(* CODESYS project SPT_Diagnostic.library
   Author: SPT
   Version: 4.0.1
   Title: SPT Diagnostic
   DefaultNamespace: SPT_Diagnostic
   Placeholder: SPT Diagnostic
   Company: Beckhoff Automation LLC

Project tree, tasks and I/O mapping:
  libraries: SPT Base Types, * (Beckhoff Automation LLC); SPT Event Logger, * (Beckhoff Automation LLC); Tc2_EtherCAT, * (Beckhoff Automation GmbH); Tc2_IoFunctions, * (Beckhoff Automation GmbH); Tc2_Standard, * (Beckhoff Automation GmbH); Tc2_System, * (Beckhoff Automation GmbH); Tc2_Utilities, * (Beckhoff Automation GmbH); Tc3_EventLogger, * (Beckhoff Automation GmbH); Tc3_Module, * (Beckhoff Automation GmbH)
  Device Diagnostic/
    DUT/
      data type ST_DeviceInfo
    function block FB_Component_Devices [ST]: Reset, CyclicLogic, CyclicLogic_EtherCat, Update, Initialize, DeviceInfo, LocalAmsNetId
  EtherCat Diagnostic/
    DUT/
      data type ST_EtherCatMaster_Command
      data type ST_EtherCatMaster_Config
      data type ST_EtherCatMaster_HMI
      data type ST_EtherCatMaster_Status
      data type ST_SyncUnitInfo
    function F_EtherCAT_VendorIDtoString [ST]
    function block FB_EtherCatMaster [ST]: CreateEvents, Monitoring, Reset, CyclicLogic, Update, GetSlaveNameByAddr, GetSyncUnitSlaveNames, LookupMasterDevState, LookupSlaveDevState, RaiseAlarmWithStringsAndFlags, RaiseWarningWithStringParameters, SlaveIsPartOfSyncUnit, FB_init, HMICommunication, Initialize, MasterState, SlaveState, EtherCatMasterInfo
    function block FB_EtherCatSyncUnits [ST]: CyclicLogic, SyncUnits, Update, LocalAmsNetId
  Interface/
    interface I_Diagnostic: Update
    interface I_EtherCatSyncUnits: SyncUnits
    interface I_SafetyBase: DependenceFB, OK, SafetyReset
    interface I_SafetyReset: Execute, PulseDuration
    interface I_SafetySimulation: SimulateSafetyDiag, SimulateSafetyState
  Project Information/
    function F_GetCompany [ST]
    function F_GetTitle [ST]
    function F_GetVersion [ST]
  Safety/
    Safety FBs Diagnostic/
      DUT/
        data type E_ComponentSafetyConnection_State
        data type E_ComponentSafetyEdm_State
        data type E_ComponentSafetyEStop_State
        data type E_ComponentSafetyGroup_Diag
        data type E_ComponentSafetyGroup_State
        data type E_ComponentSafetyMon_State
        data type E_ComponentSafetyOrAnd_State
        data type ST_SafetyStateDiag
      Reset Functionblocks/
        function block FB_SafetyResetPulse [ST]: CyclicLogic, Execute, PulseDuration
      function block FB_Component_Safety_AndOrFB [ST]: CyclicLogic, Initialize
      function block FB_Component_Safety_Base [ST]: Reset, CyclicLogic, DependenceFB, OK, SafetyReset, SimulateSafetyDiag, SimulateSafetyState, Initialize
      function block FB_Component_Safety_ConnectionFB [ST]: CreateEvents, Monitoring, Reset, CyclicLogic, Initialize
      function block FB_Component_Safety_EdmFB [ST]: CreateEvents, Monitoring, Reset, CyclicLogic, Initialize
      function block FB_Component_Safety_EstopFB [ST]: CreateEvents, Monitoring, Reset, CyclicLogic, ActiveName, Initialize
      function block FB_Component_Safety_Group [ST]: CreateEvents, Monitoring, Reset, CyclicLogic, AutoResetConnectionFaults, Initialize
      function block FB_Component_Safety_MonFB [ST]: CreateEvents, Monitoring, Reset, CyclicLogic, ActiveAlarm, ActiveName
    Safety Hardware Diagnostic/
  Version/
    global variables Global_Version
  00000000-0000-0000-0000-000000000000|LICENSE
  LICENSE
  global variables Parameter_Diagnostic
*)

// Device Diagnostic/DUT/ST_DeviceInfo
TYPE ST_DeviceInfo :
	STRUCT
		AmsNetID	   : T_AMSNETID;
		DeviceID	   : UINT;
		DeviceName	   : T_MAXSTRING;
		DeviceType	   : IODEVICETYPES;
		ipDiagnosticFB : I_Diagnostic;
	END_STRUCT
END_TYPE

// EtherCat Diagnostic/DUT/ST_EtherCatMaster_Command
TYPE ST_EtherCatMaster_Command :
	STRUCT
	END_STRUCT
END_TYPE

// EtherCat Diagnostic/DUT/ST_EtherCatMaster_Config
TYPE ST_EtherCatMaster_Config :
	STRUCT
		DeviceInfo : ST_DeviceInfo;
	END_STRUCT
END_TYPE

// EtherCat Diagnostic/DUT/ST_EtherCatMaster_HMI
TYPE ST_EtherCatMaster_HMI :
	STRUCT
		Config	: ST_EtherCatMaster_Config;
		Command : ST_EtherCatMaster_Command;
		Status	: ST_EtherCatMaster_Status;
	END_STRUCT
END_TYPE

// EtherCat Diagnostic/DUT/ST_EtherCatMaster_Status
TYPE ST_EtherCatMaster_Status :
	STRUCT
		EcSlavesState		: ARRAY[0..Parameter_Diagnostic.ETHERCAT_MASTER_SLAVE_MAX] OF ST_EcSlaveState;
		ConfiguredSlaveInfo : ARRAY[0..Parameter_Diagnostic.ETHERCAT_MASTER_SLAVE_MAX] OF ST_EcSlaveConfigData;
		EcSlaveTopologyInfo : ARRAY[0..Parameter_Diagnostic.ETHERCAT_MASTER_SLAVE_MAX] OF ST_TopologyDataEx;
	END_STRUCT
END_TYPE

// EtherCat Diagnostic/DUT/ST_SyncUnitInfo
TYPE ST_SyncUnitInfo :
	STRUCT
		Parent		   : T_MAXSTRING;
		Name		   : STRING(63);
		NumberOfSlaves : UINT;
		Slaves		   : ARRAY[1..Parameter_Diagnostic.ETHERCAT_MASTER_SYNC_UNIT_SLAVE_MAX] OF UINT;
	END_STRUCT
END_TYPE

// Safety/Safety FBs Diagnostic/DUT/E_ComponentSafetyConnection_State
{attribute 'qualified_only'}
{attribute 'strict'}
TYPE E_ComponentSafetyConnection_State : (
		Reset	   := 100,
		Session	   := 101,
		Connection := 102,
		Parameter  := 103,
		Data	   := 104,
		Shutdown   := 105,
		Deactive   := 106
	) USINT;
END_TYPE

// Safety/Safety FBs Diagnostic/DUT/E_ComponentSafetyEdm_State
{attribute 'qualified_only'}
TYPE E_ComponentSafetyEdm_State : (
		Invalid := 0,
		Stop	:= 2,
		Error	:= 4,
		Reset	:= 5,
		MonOff	:= 14,
		MonOn	:= 15
	) USINT;
END_TYPE

// Safety/Safety FBs Diagnostic/DUT/E_ComponentSafetyEStop_State
{attribute 'qualified_only'}
TYPE E_ComponentSafetyEStop_State : (
		Invalid	 := 0,
		Run		 := 1,
		Stop	 := 2,
		Safe	 := 3,
		Error	 := 4,
		Reset	 := 5,
		Start	 := 6,
		DelayOut := 7
	) USINT;
END_TYPE

// Safety/Safety FBs Diagnostic/DUT/E_ComponentSafetyGroup_Diag
{attribute 'qualified_only'}
TYPE E_ComponentSafetyGroup_Diag : (
		NoError		  := 0,
		FbError		  := 1,
		ComError	  := 2,
		ModuleError	  := 3,
		CmpError	  := 4,
		DeactiveError := 5,
		RestartError  := 6
	) UINT;
END_TYPE

// Safety/Safety FBs Diagnostic/DUT/E_ComponentSafetyGroup_State
{attribute 'qualified_only'}
TYPE E_ComponentSafetyGroup_State : (
		Invalid		 := 0,
		Run			 := 1,
		Stop		 := 2,
		Error		 := 4,
		Reset		 := 5,
		Start		 := 6,
		StopError	 := 7,
		Deactive	 := 16,
		WaitComError := 17
	) USINT;
END_TYPE

// Safety/Safety FBs Diagnostic/DUT/E_ComponentSafetyMon_State
{attribute 'qualified_only'}
TYPE E_ComponentSafetyMon_State : (
		Invalid	   := 0,
		Run		   := 1,
		Stop	   := 2,
		Safe	   := 3,
		Error	   := 4,
		Reset	   := 5,
		Start	   := 6,
		ErrorDelay := 7,
		DelayOut   := 8,
		FuncTest   := 9
	) USINT;
END_TYPE

// Safety/Safety FBs Diagnostic/DUT/E_ComponentSafetyOrAnd_State
{attribute 'qualified_only'}
TYPE E_ComponentSafetyOrAnd_State : (
		Invalid := 0,
		Run		:= 1,
		Stop	:= 2,
		Safe	:= 3
	) USINT;
END_TYPE

// Safety/Safety FBs Diagnostic/DUT/ST_SafetyStateDiag
{attribute 'pack_mode' := '1'}
TYPE ST_SafetyStateDiag :
	STRUCT
		State : USINT;
		Diag  : UINT; // **NOT PRESENT ON AND/OR FBs ** For components with USINT as Diag connection, connect first 8 Bit of UINT Diag. Inherited FB is evaluating correct length.
	END_STRUCT
END_TYPE

// Version/Global_Version
{attribute 'TcGenerated'}
{attribute 'no-analysis'}
{attribute 'linkalways'}
// This function has been automatically generated from the project information.
VAR_GLOBAL CONSTANT
	{attribute 'const_non_replaced'}
	stLibVersion_SPT_Diagnostic : ST_LibVersion := (iMajor := 4, iMinor := 0, iBuild := 1, iRevision := 0, nFlags := 0, sVersion := '4.0.1');
END_VAR

// Parameter_Diagnostic
{attribute 'qualified_only'}
VAR_GLOBAL CONSTANT
	UPDATE_TIME : TIME	:= T#500MS; // Start Diagnostic Run every xxx ms, T#0s = deactivated, update needs to manually occur via I_Diagnostic.Upadate()
	DEVICES_MAX : UDINT := 5;		// Max Devices in this System

	// EtherCat
	ETHERCAT_MASTER_START_UP_TIME		: TIME					  := T#1S; // Time to Startup EtherCat Master Diagnostic at initial startup
	ETHERCAT_MASTER_MAX					: UDINT					  := 5;	   // Max EtherCat Masters
	ETHERCAT_MASTER_SLAVE_MAX			: UDINT(1..EC_MAX_SLAVES) := 50;   // Max Slaves per EtherCat Master
	ETHERCAT_MASTER_SYNC_UNIT_MAX		: UDINT					  := 10;   // Max Count of Sync Units per Master
	ETHERCAT_MASTER_SYNC_UNIT_SLAVE_MAX : UDINT					  := 30;   // Max Count of Slaves per Sync Unit
END_VAR

// Device Diagnostic/FB_Component_Devices
{attribute 'no_explicit_call' := 'do not call this FB directly'}
FUNCTION_BLOCK FB_Component_Devices EXTENDS FB_ComponentBase IMPLEMENTS I_Diagnostic
VAR
	// System Information
	GetLocalAmsNetId : FB_GetLocalAmsNetId;
	GetDeviceIds	 : IOF_GetDeviceIDs;
	DeviceIds		 : ARRAY[0..Parameter_Diagnostic.DEVICES_MAX] OF WORD; // 0 = Device counter, 1..X = Device ID's
	GetDeviceType	 : IOF_GetDeviceType;
	GetDeviceName	 : IOF_GetDeviceName;
	GetDeviceNetId	 : IOF_GetDeviceNetId;

	// Instances of Devices
	EtherCatSyncUnits	: FB_EtherCatSyncUnits;																		  // All Sync Units in this runtime
	EtherCatMaster		: ARRAY[1..Parameter_Diagnostic.ETHERCAT_MASTER_MAX] OF FB_EtherCatMaster(EtherCatSyncUnits); //
	EtherCatMasterCount : UDINT(0..Parameter_Diagnostic.ETHERCAT_MASTER_MAX) := 0;									  // Start at 0 to identify existing during Initialzation

	// Properties
	_DeviceInfo	   : ARRAY[1..Parameter_Diagnostic.DEVICES_MAX] OF ST_DeviceInfo;
	_LocalAmsNetId : T_AmsNetId := '';

	// Alarms

	// HMI

	// Sequences
	InitializeSequence : UDINT := 0;
	DeviceNumber	   : UDINT := 1;
	i				   : UDINT := 0; // Iterator
END_VAR

VAR
	// Local
	UpdateOn	: TON;
	UpdateOff	: TON;
	RtrigUpdate : R_TRIG;
END_VAR

// Clears error flags and error IDs for this component
METHOD PUBLIC Reset : BOOL
Reset := SUPER^.Reset();
IF EtherCatMasterCount >= 1 THEN
	FOR i := 1 TO EtherCatMasterCount DO
		EtherCatMaster[i].Reset();
	END_FOR
END_IF
END_METHOD

// This method serves as the entry point for all underlying FB logic
METHOD PUBLIC CyclicLogic

// This method should be called cyclically by descendant function blocks by invoking SUPER^.CyclicLogic().  Alternatively, the contents of this method could be reimplemented entirely in which case a call to this method would not be necessary.
IF NOT _InitComplete THEN
	_InitComplete := Initialize();
	RETURN;
END_IF

// Update Toggle
IF Parameter_Diagnostic.UPDATE_TIME > T#0MS THEN
	UpdateOn(IN := NOT UpdateOff.Q, PT := Parameter_Diagnostic.UPDATE_TIME);
	UpdateOff(IN := UpdateOn.Q, PT := Parameter_Diagnostic.UPDATE_TIME);
	RtrigUpdate(CLK := UpdateOn.Q);
END_IF

// Cyclic Logics
CyclicLogic_EtherCat();
SUPER^.CyclicLogic();

// Error Status Update of all Devices
_Error := FALSE;
_Busy  := FALSE;
IF EtherCatMasterCount >= 1 THEN
	FOR i := 1 TO EtherCatMasterCount DO
		IF _CurrentAlarmSeverity < EtherCatMaster[i].CurrentAlarmSeverity THEN
			_CurrentAlarmSeverity := EtherCatMaster[i].CurrentAlarmSeverity;
		END_IF

		_Error := _Error OR EtherCatMaster[i].Error;
		_Busy  := _Busy OR EtherCatMaster[i].Busy;
		IF EtherCatMaster[i].ErrorID <> 0 AND _ErrorID = 0 THEN
			_ErrorID := EtherCatMaster[i].ErrorID;
		END_IF
	END_FOR
END_IF
END_METHOD

METHOD CyclicLogic_EtherCat
// Get all Sync Units in Runtime
EtherCatSyncUnits.LocalAmsNetId := _LocalAmsNetId;
EtherCatSyncUnits.CyclicLogic();

// Call Cyclic
IF EtherCatMasterCount >= 1 THEN
	FOR i := 1 TO EtherCatMasterCount DO
		// Update
		IF RtrigUpdate.Q THEN
			EtherCatMaster[i].Update();
		END_IF

		// Cyclic Call
		EtherCatMaster[i].CyclicLogic();
	END_FOR
END_IF
END_METHOD

METHOD Update
IF EtherCatMasterCount >= 1 THEN
	FOR i := 1 TO EtherCatMasterCount DO
		EtherCatMaster[i].Update();
	END_FOR
END_IF
END_METHOD

// Basic component initialization logic
METHOD PROTECTED Initialize : BOOL;
// This method is called by CyclicLogic() as required
VAR_INST
	AllDevicesInitialized : BOOL := FALSE;
END_VAR
Initialize := FALSE;
IF _Simulate THEN
	Initialize := SUPER^.Initialize();
	RETURN;
END_IF

// Call FBs
GetLocalAmsNetId(tTimeOut := T#1S);
GetDeviceIds(NETID := _LocalAmsNetId, TMOUT := T#1S);
GetDeviceName(NETID := _LocalAmsNetId, TMOUT := T#1S);
GetDeviceNetId(NETID := _LocalAmsNetId, TMOUT := T#1S);
GetDeviceType(NETID := _LocalAmsNetId, TMOUT := T#1S);

// Init Sequence
CASE InitializeSequence OF
	0: // Get local AmsNet-Id
		GetLocalAmsNetId.bExecute := TRUE;
		IF GetLocalAmsNetId.bBusy THEN
			InitializeSequence := InitializeSequence + 10;
		END_IF

	10: // Get local AmsNet-Id
		IF NOT GetLocalAmsNetId.bBusy AND NOT GetLocalAmsNetId.bError THEN
			_LocalAmsNetId	   := GetLocalAmsNetId.AddrString;
			InitializeSequence := InitializeSequence + 10;
		END_IF

		IF GetLocalAmsNetId.bError THEN
			_ErrorID := GetLocalAmsNetId.nErrId;
			Trace('Init Failed - GetLocalAmsNetId!');
			InitializeSequence := 999;
		END_IF

	20: // Get all Devices in this System
		GetDeviceIds.LEN	  := SIZEOF(DeviceIds);
		GetDeviceIds.DESTADDR := ADR(DeviceIds);
		GetDeviceIds.START	  := TRUE;
		IF GetDeviceIds.BUSY THEN
			GetDeviceIds.START := FALSE;
			InitializeSequence := InitializeSequence + 10;
		END_IF

	30: // Get all Devices in this System
		IF NOT GetDeviceIds.BUSY AND NOT GetDeviceIds.ERR THEN
			// Devices found
			IF (DeviceIDs[0] > 0) AND NOT _Simulate THEN
				// Map device Ids
				FOR i := 1 TO DeviceIDs[0] DO
					IF i <= Parameter_Diagnostic.DEVICES_MAX THEN
						_DeviceInfo[i].DeviceID := DeviceIDs[i];
					ELSE
						Trace('Init Failed - find IO Devices, Diagnostic, not enough Devices foreseen! Increase DEVICES_MAX');
						InitializeSequence := 999;
						EXIT;
					END_IF
				END_FOR

				InitializeSequence := InitializeSequence + 10;
			ELSE
				_Simulate		   := TRUE; // No devices found = activate simulation mode
				InitializeSequence := 1000;
			END_IF
		END_IF

		IF GetDeviceIds.ERR THEN
			_ErrorID := GetDeviceIds.ERRID;
			Trace('Init Failed - GetDeviceIds!');
			InitializeSequence := 999;
		END_IF

	40: // Get Device Names
		GetDeviceName.DEVICEID := DeviceIDs[DeviceNumber];
		GetDeviceName.START	   := TRUE;
		IF GetDeviceName.BUSY THEN
			GetDeviceName.START := FALSE;
			InitializeSequence	:= InitializeSequence + 10;
		END_IF

	50: // Get Device Names
		IF NOT GetDeviceName.BUSY AND NOT GetDeviceName.ERR THEN
			// Next Device
			_DeviceInfo[DeviceNumber].DeviceName := GetDeviceName.DEVICENAME;
			DeviceNumber						 := DeviceNumber + 1;
			IF (DeviceIDs[DeviceNumber] <> 0) THEN
				InitializeSequence := InitializeSequence - 10;
			ELSE
				DeviceNumber	   := 1;
				InitializeSequence := InitializeSequence + 10;
			END_IF
		END_IF

		IF GetDeviceName.ERR THEN
			_ErrorID := GetDeviceName.ERRID;
			Trace('Init Failed - GetDeviceName!');
			InitializeSequence := 999;
		END_IF

	60: // Get Device NetIds
		GetDeviceNetId.DEVICEID := DeviceIDs[DeviceNumber];
		GetDeviceNetId.START	:= TRUE;
		IF GetDeviceNetId.BUSY THEN
			GetDeviceNetId.START := FALSE;
			InitializeSequence	 := InitializeSequence + 10;
		END_IF

	70: // Get Device NetIds
		IF NOT GetDeviceNetId.BUSY AND NOT GetDeviceNetId.ERR THEN
			// Next Device
			_DeviceInfo[DeviceNumber].AmsNetID := GetDeviceNetId.DeviceNetId;
			DeviceNumber					   := DeviceNumber + 1;
			IF (DeviceIDs[DeviceNumber] <> 0) THEN
				InitializeSequence := InitializeSequence - 10;
			ELSE
				DeviceNumber	   := 1;
				InitializeSequence := InitializeSequence + 10;
			END_IF
		END_IF

		IF GetDeviceNetId.ERR THEN
			_ErrorID := GetDeviceNetId.ERRID;
			Trace('Init Failed - GetDeviceNetId!');
			InitializeSequence := 999;
		END_IF

	80: // Get Device Types
		GetDeviceType.DEVICEID := DeviceIDs[DeviceNumber];
		GetDeviceType.START	   := TRUE;
		IF GetDeviceType.BUSY THEN
			GetDeviceType.START := FALSE;
			InitializeSequence	:= InitializeSequence + 10;
		END_IF

	90: // Get Device Types
		IF NOT GetDeviceType.BUSY AND NOT GetDeviceType.ERR THEN
			// Next Device
			_DeviceInfo[DeviceNumber].DeviceType := GetDeviceType.IODeviceType;
			DeviceNumber						 := DeviceNumber + 1;
			IF (DeviceIDs[DeviceNumber] <> 0) THEN
				InitializeSequence := InitializeSequence - 10;
			ELSE
				DeviceNumber	   := 1;
				InitializeSequence := InitializeSequence + 10;
			END_IF
		END_IF

		IF GetDeviceType.ERR THEN
			_ErrorID := GetDeviceType.ERRID;
			Trace('Init Failed - GetDeviceType!');
			InitializeSequence := 999;
		END_IF

	100: // Initalize all Devices found
		FOR i := 1 TO DeviceIDs[0] DO
			CASE DeviceInfo[i].DeviceType OF
				IODEVICETYPES.IODEVICETYPE_ETHERCAT:
					EtherCatMasterCount := EtherCatMasterCount + 1;
					IF EtherCatMasterCount <= Parameter_Diagnostic.ETHERCAT_MASTER_MAX THEN
						EtherCatMaster[EtherCatMasterCount].EtherCatMasterInfo REF= _DeviceInfo[i];
						EtherCatMaster[EtherCatMasterCount].Name			   := DeviceInfo[i].DeviceName;
						DeviceInfo[i].ipDiagnosticFB						   := EtherCatMaster[EtherCatMasterCount];
					ELSE
						Trace('Init Failed - not enough EtherCat Master Diagnostics Instances! Increase ETHERCAT_MASTER_MAX');
						InitializeSequence := 999;
					END_IF

			ELSE
				Trace(CONCAT('Warning - Device Diagnostics for this Device does not exist! ', DeviceInfo[i].DeviceName));
			END_CASE
		END_FOR

		// No error during initialization
		IF InitializeSequence <> 999 THEN
			InitializeSequence := InitializeSequence + 10;
		END_IF

	110: // Initalize all Devices found
		AllDevicesInitialized := TRUE;

		// Init all EtherCat Master Devices
		IF EtherCatMasterCount >= 1 THEN
			FOR i := 1 TO EtherCatMasterCount DO
				EtherCatMaster[i].CyclicLogic();
				AllDevicesInitialized := AllDevicesInitialized AND EtherCatMaster[i].InitComplete;
			END_FOR
		END_IF

		IF AllDevicesInitialized THEN
			InitializeSequence := 1000;
		END_IF

	1000: // Initialize the Base
		IF SUPER^.Initialize() THEN
			Initialize := TRUE;
			_Error	   := FALSE;
			_Busy	   := FALSE;
		END_IF

	999:
		_Error := TRUE;
		_Busy  := FALSE;
END_CASE
END_METHOD

{analysis -29}
PROPERTY DeviceInfo : REFERENCE TO ARRAY[1..Parameter_Diagnostic.DEVICES_MAX] OF ST_DeviceInfo
GET
DeviceInfo REF= _DeviceInfo;
END_GET
END_PROPERTY

PROPERTY LocalAmsNetId : T_AmsNetId
GET
LocalAmsNetId := _LocalAmsNetId;
END_GET
END_PROPERTY

END_FUNCTION_BLOCK

// Interface/I_Diagnostic
INTERFACE I_Diagnostic EXTENDS I_BaseFB

METHOD Update
VAR_INPUT
END_VAR
END_METHOD

END_INTERFACE

// EtherCat Diagnostic/FB_EtherCatSyncUnits
{attribute 'no_explicit_call' := 'do not call this FB directly'}
FUNCTION_BLOCK FB_EtherCatSyncUnits EXTENDS FB_CyclicFB IMPLEMENTS I_EtherCatSyncUnits
VAR
	(* Sequence *)
	SyncUnitSequence : UINT;

	(* Local *)
	GetSyncUnitOids			  : ADSRDWRT;
	GetAllSyncUnitSlaveAddr	  : FB_EcGetAllSyncUnitSlaveAddr;
	ipSyncUnitComObject		  : ITComObject;
	ipSyncUnitParentComObject : ITComObject;
	SyncUnitCount			  : DWORD;
	i						  : DWORD; // Iterator
	SyncUnitParentOid		  : OTCID;
	SyncUnitOids			  : ARRAY[1..Parameter_Diagnostic.ETHERCAT_MASTER_SYNC_UNIT_MAX] OF OTCID;

	(* Properties *)
	_SyncUnits	   : ARRAY[1..Parameter_Diagnostic.ETHERCAT_MASTER_SYNC_UNIT_MAX] OF ST_SyncUnitInfo;
	_LocalAmsNetId : T_AmsNetId;
END_VAR

VAR CONSTANT
	SYNC_UNIT_CLASS_ID : CLSID := STRING_TO_GUID('03020004-0000-0000-F000-000000000064');
END_VAR

METHOD PUBLIC CyclicLogic
VAR_INST
	tempName		 : STRING(63);
	SyncUnitIterator : UINT := 1;
END_VAR
{analysis -19}
{analysis -07}

// Call FBs
GetSyncUnitOids(NETID := _LocalAmsNetId);
GetAllSyncUnitSlaveAddr(sNetId := _LocalAmsNetId);

// Sequence
CASE SyncUnitSequence OF
	0: // Wait for start
		GetSyncUnitOids.WRTRD			 := FALSE;
		GetAllSyncUnitSlaveAddr.bExecute := FALSE;
		SyncUnitIterator				 := 1;

	10: // Get Sync Unit Count

		// Reset for restart
		_Error	 := FALSE;
		_ErrorID := 0;

		// Get Sync Unit Count
		GetSyncUnitOids.PORT	 := 10;
		GetSyncUnitOids.IDXGRP	 := 16#201;
		GetSyncUnitOids.IDXOFFS	 := 16#01;
		GetSyncUnitOids.WRITELEN := SIZEOF(SYNC_UNIT_CLASS_ID);
		GetSyncUnitOids.SRCADDR	 := ADR(SYNC_UNIT_CLASS_ID);
		GetSyncUnitOids.READLEN	 := SIZEOF(SyncUnitCount);
		GetSyncUnitOids.DESTADDR := ADR(SyncUnitCount);
		GetSyncUnitOids.WRTRD	 := TRUE;
		IF GetSyncUnitOids.BUSY THEN
			SyncUnitSequence := SyncUnitSequence + 10;
		END_IF

	20: // Get Sync Unit Count
		IF NOT GetSyncUnitOids.BUSY AND NOT GetSyncUnitOids.ERR THEN
			// Byte Adjustment
			SyncUnitCount		  := SyncUnitCount / 4;
			GetSyncUnitOids.WRTRD := FALSE;
			IF SyncUnitCount <= Parameter_Diagnostic.ETHERCAT_MASTER_SYNC_UNIT_MAX THEN // Check configuration and space
				IF SyncUnitCount > 0 THEN												// Only if Sync Unit exist - run diag
					SyncUnitSequence := SyncUnitSequence + 10;
				ELSE
					SyncUnitSequence := 0;
				END_IF
			ELSE
				SyncUnitSequence := 999;
				_ErrorID		 := SyncUnitCount;
				Trace('FB_EtherCatSyncUnits - not enough Sync Units foreseen! Increase ETHERCAT_MASTER_SYNC_UNIT_MAX');
			END_IF
		END_IF

		IF GetSyncUnitOids.ERR THEN
			_ErrorID		 := GetSyncUnitOids.ERRID;
			SyncUnitSequence := 999;
		END_IF

	30: // Get Sync Unit Oids
		GetSyncUnitOids.PORT	 := 10;
		GetSyncUnitOids.IDXGRP	 := 16#201;
		GetSyncUnitOids.IDXOFFS	 := 16#02;
		GetSyncUnitOids.WRITELEN := SIZEOF(SYNC_UNIT_CLASS_ID);
		GetSyncUnitOids.SRCADDR	 := ADR(SYNC_UNIT_CLASS_ID);
		GetSyncUnitOids.READLEN	 := (SIZEOF(OTCID) * SyncUnitCount);
		GetSyncUnitOids.DESTADDR := ADR(SyncUnitOids);
		GetSyncUnitOids.WRTRD	 := TRUE;
		IF GetSyncUnitOids.BUSY THEN
			SyncUnitSequence := SyncUnitSequence + 10;
		END_IF

	40: // Get Sync Unit Oids
		IF NOT GetSyncUnitOids.BUSY AND NOT GetSyncUnitOids.ERR THEN
			GetSyncUnitOids.WRTRD := FALSE;
			SyncUnitSequence	  := SyncUnitSequence + 10;
		END_IF

		IF GetSyncUnitOids.ERR THEN
			_ErrorID		 := GetSyncUnitOids.ERRID;
			SyncUnitSequence := 999;
		END_IF

	50: // Get EtherCat Master and Name of Sync Unit
		FOR i := 1 TO SyncUnitCount DO
			// Get Sync Unit
			FW_ObjMgr_GetObjectInstance(SyncUnitOids[i], TC_GLOBAL_IID_LIST.IID_ITComObject, ADR(ipSyncUnitComObject));
			IF ipSyncUnitComObject <> 0 THEN
				ipSyncUnitComObject.TcGetObjectName(objName := ADR(_SyncUnits[i].Name), nameLen := SIZEOF(_SyncUnits[i].Name));
				F_EcGetSyncUnitName(SyncUnitOids[i], sSyncUnitName => tempName);
				tempName		   := CONCAT(tempName, ' - ');
				_SyncUnits[i].Name := CONCAT(tempName, _SyncUnits[i].Name);

				// Get Parent
				ipSyncUnitComObject.TcGetParentObjId(SyncUnitParentOid);
				FW_ObjMgr_GetObjectInstance(SyncUnitParentOid, TC_GLOBAL_IID_LIST.IID_ITComObject, ADR(ipSyncUnitParentComObject));
				IF ipSyncUnitParentComObject <> 0 THEN
					ipSyncUnitParentComObject.TcGetObjectName(objName := ADR(_SyncUnits[i].Parent), nameLen := SIZEOF(_SyncUnits[i].Parent));
					FW_SafeRelease(pipUnk := ADR(ipSyncUnitParentComObject));
				END_IF

				FW_SafeRelease(pipUnk := ADR(ipSyncUnitComObject));
			END_IF
		END_FOR

		SyncUnitSequence := SyncUnitSequence + 10;

	60: // Get all sync Unit Slaves 
		IF SyncUnitIterator > Parameter_Diagnostic.ETHERCAT_MASTER_SYNC_UNIT_MAX THEN
			SyncUnitSequence := 0; // All Sync units searched
		ELSE
			IF SyncUnitOids[SyncUnitIterator] = 0 THEN
				SyncUnitSequence := 0; // Done
			ELSE
				GetAllSyncUnitSlaveAddr.nObjectId := SyncUnitOids[SyncUnitIterator];
				GetAllSyncUnitSlaveAddr.pAddrBuf  := ADR(_SyncUnits[SyncUnitIterator].Slaves);
				GetAllSyncUnitSlaveAddr.cbBufLen  := SIZEOF(_SyncUnits[SyncUnitIterator].Slaves);
				GetAllSyncUnitSlaveAddr.bExecute  := TRUE;
				IF GetAllSyncUnitSlaveAddr.bBusy THEN
					GetAllSyncUnitSlaveAddr.bExecute := FALSE;
					SyncUnitSequence				 := SyncUnitSequence + 10;
				END_IF
			END_IF
		END_IF

	70: // Get all sync Unit Slaves
		IF NOT GetAllSyncUnitSlaveAddr.bBusy AND NOT GetAllSyncUnitSlaveAddr.bError THEN
			_SyncUnits[SyncUnitIterator].NumberOfSlaves := GetAllSyncUnitSlaveAddr.nSlaves;
			SyncUnitIterator							:= SyncUnitIterator + 1;
			IF _SyncUnits[SyncUnitIterator].NumberOfSlaves <= Parameter_Diagnostic.ETHERCAT_MASTER_SYNC_UNIT_SLAVE_MAX THEN
				SyncUnitSequence := SyncUnitSequence - 10;
			ELSE
				SyncUnitSequence := 999;
				_ErrorID		 := _SyncUnits[SyncUnitIterator].NumberOfSlaves;
				Trace('FB_EtherCatSyncUnits - not enough slaves per Sync Units foreseen! Increase ETHERCAT_MASTER_SYNC_UNIT_SLAVE_MAX');
			END_IF
		END_IF

		IF GetAllSyncUnitSlaveAddr.bError THEN
			_ErrorID		 := GetAllSyncUnitSlaveAddr.nErrId;
			SyncUnitSequence := 999;
		END_IF

	999: // Error
		SyncUnitSequence := 0;
		_Error			 := TRUE;
		Trace('FB_EtherCatSyncUnits - Error get Sync Units Sequence!');
END_CASE

_Busy := SyncUnitSequence <> 0;
END_METHOD

PROPERTY SyncUnits : REFERENCE TO ARRAY[1..Parameter_Diagnostic.ETHERCAT_MASTER_SYNC_UNIT_MAX] OF ST_SyncUnitInfo
GET
SyncUnits REF= _SyncUnits;
END_GET
END_PROPERTY

METHOD Update
IF NOT _Busy THEN
	SyncUnitSequence := 10;
END_IF
END_METHOD

PROPERTY LocalAmsNetId : T_AmsNetId
SET
_LocalAmsNetId := LocalAmsNetId;
END_SET
END_PROPERTY

END_FUNCTION_BLOCK

// Interface/I_EtherCatSyncUnits
INTERFACE I_EtherCatSyncUnits EXTENDS I_Diagnostic

PROPERTY SyncUnits : REFERENCE TO ARRAY[1..Parameter_Diagnostic.ETHERCAT_MASTER_SYNC_UNIT_MAX] OF ST_SyncUnitInfo
GET
END_GET
END_PROPERTY

END_INTERFACE

// EtherCat Diagnostic/FB_EtherCatMaster
{attribute 'no_explicit_call' := 'do not call this FB directly'}
FUNCTION_BLOCK FB_EtherCatMaster EXTENDS FB_ComponentBase IMPLEMENTS I_Diagnostic
VAR
	(* Internal Variables *)
	EcGetMasterDevState	 : FB_EcGetMasterDevState;
	GetSlaveTopologyInfo : FB_EcGetSlaveTopologyInfo;
	EcGetAllSlaveStates	 : FB_EcGetAllSlaveStates;
	GetConfiguredSlaves	 : FB_EcGetConfSlaves;
	EcSlavesState		 : ARRAY[0..Parameter_Diagnostic.ETHERCAT_MASTER_SLAVE_MAX] OF ST_EcSlaveState;
	ConfiguredSlaveInfo	 : ARRAY[0..Parameter_Diagnostic.ETHERCAT_MASTER_SLAVE_MAX] OF ST_EcSlaveConfigData;
	EcSlaveTopologyInfo	 : ARRAY[0..Parameter_Diagnostic.ETHERCAT_MASTER_SLAVE_MAX] OF ST_TopologyDataEx;
	SyncUnits			 : REFERENCE TO ARRAY[1..Parameter_Diagnostic.ETHERCAT_MASTER_SYNC_UNIT_MAX] OF ST_SyncUnitInfo;
	MasterDevState		 : WORD;
	SlaveCount			 : UINT;
	CfgSlaveCount		 : UINT;

	(* Properties *)
	_EtherCatMasterInfo : REFERENCE TO ST_DeviceInfo;

	(* HMI *)
	EtherCatMaster_HMI : ST_EtherCatMaster_HMI;

	(* Sync Units *)
	ipEtherCatSyncUnits : I_EtherCatSyncUnits;

	(* Sequence *)
	SlaveSeq	: UINT;
	MasterSeq	: UINT;
	SyncUnitSeq : UINT;

	(* Alarms *)
	MasterAlarms	 : ARRAY[1..MASTER_ALARM_COUNT] OF FB_TcAlarm;
	SlaveErrors		 : ARRAY[0..Parameter_Diagnostic.ETHERCAT_MASTER_SLAVE_MAX] OF FB_TcAlarm;
	SlaveWarnings	 : ARRAY[0..Parameter_Diagnostic.ETHERCAT_MASTER_SLAVE_MAX] OF FB_TcAlarm;
	SyncUnitWarnings : ARRAY[1..Parameter_Diagnostic.ETHERCAT_MASTER_SYNC_UNIT_MAX] OF FB_TcAlarm;
END_VAR

VAR CONSTANT
	MASTER_ALARM_COUNT : UDINT := 3;
	STRING_LEN		   : INT   := 80;
END_VAR

METHOD PROTECTED CreateEvents
// This method is called by Initialize() as required
VAR_INST
	tempName   : STRING;
	SourceInfo : FB_TcSourceInfo;
	i		   : UDINT;
END_VAR
F_CreateAllEventsInClass(Alarms		:= MasterAlarms,
						 ClassSize	:= SIZEOF(TC_EVENTS.EtherCatMaster),
						 pInitEvent := ADR(TC_EVENTS.EtherCatMaster.InitReferenceEvent),
						 Prefix		:= Name);

SUPER^.CreateEvents();

// Create SyncUnit and Slave Alarms
FOR i := 0 TO Parameter_Diagnostic.ETHERCAT_MASTER_SLAVE_MAX DO
	SourceInfo.sName := CONCAT(CONCAT(THIS^.Name, ' - '), ConfiguredSlaveInfo[i].sName);
	SlaveErrors[i].CreateEx(stEventEntry := TC_EVENTS.EtherCatSlave.SlaveError, 0, SourceInfo);
	SlaveWarnings[i].CreateEx(stEventEntry := TC_EVENTS.EtherCatSlave.SlaveWarning, 0, SourceInfo);
END_FOR

FOR i := 1 TO Parameter_Diagnostic.ETHERCAT_MASTER_SYNC_UNIT_MAX DO
	SourceInfo.sName := CONCAT(CONCAT(THIS^.Name, ' - '), ConfiguredSlaveInfo[i].sName);
	SyncUnitWarnings[i].CreateEx(stEventEntry := TC_EVENTS.SyncUnit.SyncUnitWarning, 0, SourceInfo);
END_FOR
END_METHOD

// Provides basic error detection and event handling for this component
METHOD PROTECTED Monitoring
// This method is called cyclically by CyclicLogic()
VAR_INST
	Error1 : BOOL;
	Error2 : BOOL;
	Error3 : BOOL;
END_VAR
SUPER^.Monitoring();

(* EtherCat Master Messages *)

// Raised in Master Sequence

(* EtherCat Slave Messages *)

// Raised in Slave Sequence

(* Alarm Severity of EtherCat Master Device *)
_CurrentAlarmSeverity := F_GetMaxSeverityRaised(Alarms := MasterAlarms, CurrentSeverity := _CurrentAlarmSeverity);
_CurrentAlarmSeverity := F_GetMaxSeverityRaised(Alarms := SlaveErrors, CurrentSeverity := _CurrentAlarmSeverity);
_CurrentAlarmSeverity := F_GetMaxSeverityRaised(Alarms := SlaveWarnings, CurrentSeverity := _CurrentAlarmSeverity);
_CurrentAlarmSeverity := F_GetMaxSeverityRaised(Alarms := SyncUnitWarnings, CurrentSeverity := _CurrentAlarmSeverity);
END_METHOD

// Clears error flags and error IDs for this component
METHOD PUBLIC Reset : BOOL
F_ClearAllEventsInClass(MasterAlarms);
F_ClearAllEventsInClass(SlaveErrors);
F_ClearAllEventsInClass(SlaveWarnings);
F_ClearAllEventsInClass(SyncUnitWarnings);
SlaveSeq  := 0;
MasterSeq := 0;
_Error	  := FALSE;
_ErrorID  := 0;
_Busy	  := FALSE;
Reset	  := SUPER^.Reset();
END_METHOD

// This method serves as the entry point for all underlying FB logic
METHOD PUBLIC CyclicLogic

// This method should be called cyclically by descendant function blocks by invoking SUPER^.CyclicLogic().  Alternatively, the contents of this method could be reimplemented entirely in which case a call to this method would not be necessary.
IF NOT _InitComplete THEN
	_InitComplete := Initialize();
	RETURN;
END_IF

(* Main Component Signals *)
IF _Simulate THEN
	_Busy	 := FALSE;
	_Error	 := FALSE;
	_ErrorID := 0;
ELSE
	// Master State
	MasterState();

	// Slave State
	SlaveState();

	// Super
	_Busy := SlaveSeq <> 0 OR MasterSeq <> 0; // Sequence running
	SUPER^.CyclicLogic();
END_IF
END_METHOD

METHOD Update
IF NOT _Busy THEN
	// Start Master and Slave Diagnostics Sequence
	MasterSeq := 10;
	SlaveSeq  := 10;
END_IF
END_METHOD

METHOD PRIVATE GetSlaveNameByAddr : STRING(31)
VAR_INPUT
	Addr : UINT;
END_VAR

VAR_INST
	Slave : UDINT;
END_VAR
GetSlaveNameByAddr := '';
FOR Slave := 0 TO Parameter_Diagnostic.ETHERCAT_MASTER_SLAVE_MAX DO
	IF ConfiguredSlaveInfo[Slave].nAddr = Addr THEN
		GetSlaveNameByAddr := ConfiguredSlaveInfo[Slave].sName;
		RETURN;
	END_IF
END_FOR
END_METHOD

METHOD PRIVATE GetSyncUnitSlaveNames
VAR_INPUT
	SyncUnit : ST_SyncUnitInfo;
END_VAR

VAR_INST
	i						  : UDINT;
	j						  : UDINT;
	TempSlavesInSyncUnitPartA : STRING;
	TempSlavesInSyncUnitPartB : STRING;
	TempSlaveMessage		  : STRING;
END_VAR

VAR_OUTPUT
	SlavesInSyncUnitPartA : STRING;
	SlavesInSyncUnitPartB : STRING;
END_VAR
TempSlavesInSyncUnitPartA := '';
TempSlavesInSyncUnitPartB := '';
FOR i := 1 TO Parameter_Diagnostic.ETHERCAT_MASTER_SYNC_UNIT_SLAVE_MAX DO
	FOR j := 1 TO Parameter_Diagnostic.ETHERCAT_MASTER_SLAVE_MAX DO
		IF SyncUnit.Slaves[i] <> 0 THEN
			IF SyncUnit.Slaves[i] = ConfiguredSlaveInfo[j].nAddr THEN
				IF LEN(ConfiguredSlaveInfo[j].sName) > 0 THEN
					TempSlaveMessage := CONCAT(ConfiguredSlaveInfo[j].sName, ', ');
					IF (LEN(TempSlaveMessage) + LEN(TempSlavesInSyncUnitPartA)) <= STRING_LEN THEN
						TempSlavesInSyncUnitPartA := CONCAT(TempSlavesInSyncUnitPartA, TempSlaveMessage);
					ELSIF (LEN(TempSlaveMessage) + LEN(TempSlavesInSyncUnitPartB)) <= STRING_LEN THEN
						TempSlavesInSyncUnitPartB := CONCAT(TempSlavesInSyncUnitPartB, TempSlaveMessage);
					END_IF
				END_IF
			END_IF
		END_IF
	END_FOR
END_FOR

SlavesInSyncUnitPartA := TempSlavesInSyncUnitPartA;
SlavesInSyncUnitPartB := TempSlavesInSyncUnitPartB;
END_METHOD

METHOD PROTECTED LookupMasterDevState : STRING
VAR_INPUT
	State : UINT;
END_VAR

VAR_OUTPUT
	TypeError	: BOOL;
	TypeWarning : BOOL;
END_VAR
TypeError	:= FALSE;
TypeWarning := FALSE;
IF State.0 THEN
	TypeError			 := TRUE;
	LookupMasterDevState := 'Link error';
ELSIF State.1 THEN
	TypeError			 := TRUE;
	LookupMasterDevState := 'I/O locked after link error (I/O reset required)';
ELSIF State.2 THEN
	TypeError			 := TRUE;
	LookupMasterDevState := 'Link error (redundancy adapter)';
ELSIF State.3 THEN
	TypeError			 := TRUE;
	LookupMasterDevState := 'Missing one frame (redundancy mode)';
ELSIF State.4 THEN
	TypeError			 := TRUE;
	LookupMasterDevState := 'Out of send resources (I/O reset required)';
ELSIF State.5 THEN
	TypeError			 := TRUE;
	LookupMasterDevState := 'Watchdog triggered';
ELSIF State.6 THEN
	TypeError			 := TRUE;
	LookupMasterDevState := 'Ethernet driver (miniport) NOT found';
ELSIF State.7 THEN
	TypeWarning			 := TRUE;
	LookupMasterDevState := 'I/O reset active';
ELSIF State.8 THEN
	TypeWarning			 := TRUE;
	LookupMasterDevState := 'At least one device in INIT state';
ELSIF State.9 THEN
	TypeWarning			 := TRUE;
	LookupMasterDevState := 'At least one device in PRE-OP state';
ELSIF State.10 THEN
	TypeWarning			 := TRUE;
	LookupMasterDevState := 'At least one device in SAFE-OP state';
ELSIF State.11 THEN
	TypeWarning			 := TRUE;
	LookupMasterDevState := 'At least one device indicates an error state';
ELSIF State.12 THEN
	TypeError			 := TRUE;
	LookupMasterDevState := 'DC not in sync';
ELSE
	TypeWarning			 := TRUE;
	LookupMasterDevState := 'State not found';
END_IF
END_METHOD

METHOD PROTECTED LookupSlaveDevState : STRING
VAR_INPUT
	Slave : UDINT;
END_VAR

VAR_INST
	DiagByte				: BYTE;
	BitMaskDiag				: BYTE := 16#0F;
	tempLookupSlaveDevState : STRING;
END_VAR
//_____________________________________________________________________________________________________

(* State *)
BitMaskDiag := 16#0F;
DiagByte	:= EcSlavesState[Slave].deviceState AND BitMaskDiag;
CASE DiagByte OF
	EC_DEVICE_STATE_INIT:
		tempLookupSlaveDevState := 'Init';

	EC_DEVICE_STATE_PREOP:
		tempLookupSlaveDevState := 'Pre-op';

	EC_DEVICE_STATE_BOOTSTRAP:
		tempLookupSlaveDevState := 'Boot';

	EC_DEVICE_STATE_SAFEOP:
		tempLookupSlaveDevState := 'Safe-op';

	EC_DEVICE_STATE_OP:
		tempLookupSlaveDevState := 'OP';

ELSE
	tempLookupSlaveDevState := '';
END_CASE

(* Additional State Bits *)
IF EcSlavesState[Slave].deviceState.4 THEN // EC_DEVICE_STATE_ERROR
	tempLookupSlaveDevState := CONCAT(tempLookupSlaveDevState, ' - ');
	tempLookupSlaveDevState := CONCAT(tempLookupSlaveDevState, 'State machine error in the EtherCAT slave');
END_IF

IF EcSlavesState[Slave].deviceState.5 THEN // EC_DEVICE_STATE_INVALID_VPRS
	tempLookupSlaveDevState := CONCAT(tempLookupSlaveDevState, ' - ');
	tempLookupSlaveDevState := CONCAT(tempLookupSlaveDevState, 'Invalid vendor ID');
END_IF

IF EcSlavesState[Slave].deviceState.6 THEN // EC_DEVICE_STATE_INITCMD_ERROR
	tempLookupSlaveDevState := CONCAT(tempLookupSlaveDevState, ' - ');
	tempLookupSlaveDevState := CONCAT(tempLookupSlaveDevState, 'Error during sending of initialization commands');
END_IF

IF EcSlavesState[Slave].deviceState.7 THEN // EC_DEVICE_STATE_DISABLED
	tempLookupSlaveDevState := CONCAT(tempLookupSlaveDevState, ' - ');
	tempLookupSlaveDevState := CONCAT(tempLookupSlaveDevState, 'Slave is disabled');
END_IF

//_____________________________________________________________________________________________________

(* Link States *)
IF EcSlavesState[Slave].linkState.0 THEN // EC_LINK_STATE_NOT_PRESENT
	tempLookupSlaveDevState := CONCAT(tempLookupSlaveDevState, ' - ');
	tempLookupSlaveDevState := CONCAT(tempLookupSlaveDevState, 'No EtherCAT communication with the EtherCAT slave');
END_IF

IF EcSlavesState[Slave].linkState.1 THEN // EC_LINK_STATE_LINK_WITHOUT_COMM
	tempLookupSlaveDevState := CONCAT(tempLookupSlaveDevState, ' - ');
	tempLookupSlaveDevState := CONCAT(tempLookupSlaveDevState, 'Error AT port X');
END_IF

IF EcSlavesState[Slave].linkState.2 THEN // EC_LINK_STATE_MISSING_LINK
	tempLookupSlaveDevState := CONCAT(tempLookupSlaveDevState, ' - ');
	tempLookupSlaveDevState := CONCAT(tempLookupSlaveDevState, 'Missing link AT port X');
END_IF

IF EcSlavesState[Slave].linkState.3 THEN // EC_LINK_STATE_ADDITIONAL_LINK
	tempLookupSlaveDevState := CONCAT(tempLookupSlaveDevState, ' - ');
	tempLookupSlaveDevState := CONCAT(tempLookupSlaveDevState, 'Additional link AT port X');
END_IF

(* Additional State Bits *)
IF EcSlavesState[Slave].linkState.4 THEN // EC_LINK_STATE_PORT_A
	tempLookupSlaveDevState := CONCAT(tempLookupSlaveDevState, ' - ');
	tempLookupSlaveDevState := CONCAT(tempLookupSlaveDevState, 'Port 0');
END_IF

IF EcSlavesState[Slave].linkState.5 THEN // EC_LINK_STATE_PORT_B
	tempLookupSlaveDevState := CONCAT(tempLookupSlaveDevState, ' - ');
	tempLookupSlaveDevState := CONCAT(tempLookupSlaveDevState, 'Port 1');
END_IF

IF EcSlavesState[Slave].linkState.6 THEN // EC_LINK_STATE_PORT_C
	tempLookupSlaveDevState := CONCAT(tempLookupSlaveDevState, ' - ');
	tempLookupSlaveDevState := CONCAT(tempLookupSlaveDevState, 'Port 2');
END_IF

IF EcSlavesState[Slave].linkState.7 THEN // EC_LINK_STATE_PORT_D
	tempLookupSlaveDevState := CONCAT(tempLookupSlaveDevState, ' - ');
	tempLookupSlaveDevState := CONCAT(tempLookupSlaveDevState, 'Port 3');
END_IF

LookupSlaveDevState := tempLookupSlaveDevState;
END_METHOD

METHOD PRIVATE RaiseAlarmWithStringsAndFlags
VAR_INPUT
	Alarm	 : FB_TcAlarm; // Alarm to be raised
	String_1 : STRING;
	String_2 : STRING;
	String_3 : STRING;
END_VAR
IF NOT Alarm.bRaised THEN
	F_RaiseAlarmWithStringsAndFlags(Alarm	  := Alarm,
									ErrorFlag := _Error,
									ErrorID	  := _ErrorID,
									String_1  := String_1,
									String_2  := String_2,
									String_3  := String_3);
END_IF
END_METHOD

METHOD PRIVATE RaiseWarningWithStringParameters
VAR_INPUT
	Warning	 : FB_TcAlarm; // Alarm to be raised
	String_1 : STRING;
	String_2 : STRING;
	String_3 : STRING;
END_VAR
IF NOT Warning.bRaised THEN
	F_RaiseAlarmWithStringParameters(Alarm	  := Warning,
									 String_1 := String_1,
									 String_2 := String_2,
									 String_3 := String_3);
END_IF
END_METHOD

METHOD PRIVATE SlaveIsPartOfSyncUnit : BOOL
VAR_INPUT
	SlaveAddr : UINT;
	SyncUnit  : ST_SyncUnitInfo;
END_VAR

VAR_INST
	i : UDINT;
END_VAR
SlaveIsPartOfSyncUnit := FALSE;
FOR i := 1 TO Parameter_Diagnostic.ETHERCAT_MASTER_SYNC_UNIT_SLAVE_MAX DO
	IF SyncUnit.Slaves[i] = SlaveAddr THEN
		SlaveIsPartOfSyncUnit := TRUE;
		RETURN;
	END_IF
END_FOR
END_METHOD

METHOD FB_init : BOOL
VAR_INPUT
	bInitRetains	  : BOOL; // if TRUE, the retain variables are initialized (warm start / cold start)
	bInCopyCode		  : BOOL; // if TRUE, the instance afterwards gets moved into the copy code (online change)
	EtherCatSyncUnits : I_EtherCatSyncUnits;
END_VAR
IF EtherCatSyncUnits <> 0 THEN
	ipEtherCatSyncUnits := EtherCatSyncUnits;
END_IF
END_METHOD

// Provides interlocks for HMI control and updates HMI status information for this component
METHOD PROTECTED HMICommunication

// This method is called cyclically by CyclicLogic()
SUPER^.HMICommunication();

// Device Info
EtherCatMaster_HMI.Config.DeviceInfo := _EtherCatMasterInfo;

// Status
EtherCatMaster_HMI.Status.EcSlavesState		  := EcSlavesState;
EtherCatMaster_HMI.Status.ConfiguredSlaveInfo := ConfiguredSlaveInfo;
EtherCatMaster_HMI.Status.EcSlaveTopologyInfo := EcSlaveTopologyInfo;
END_METHOD

// Basic component initialization logic
METHOD PROTECTED Initialize : BOOL;
VAR_INST
	InitializeSequence : UINT := 0;
	Size			   : UDINT;
	StartupTime		   : TON;
END_VAR

// This method is called by CyclicLogic() as required
{analysis -19}
Initialize := FALSE;
IF NOT __ISVALIDREF(_EtherCatMasterInfo) THEN
	_Error := TRUE;
	Trace('Init Failed - EtherCatMasterInfo not set in EtherCat Master Component!');
END_IF

IF ipEtherCatSyncUnits = 0 THEN
	_Error := TRUE;
	Trace('Init Failed - EtherCatSyncUnits not set in constructor!');
END_IF

IF _Error THEN
	RETURN;
END_IF

IF _Simulate THEN
	Initialize := SUPER^.Initialize();
	RETURN;
END_IF

// Get all Slaves
GetConfiguredSlaves(sNetId				:= _EtherCatMasterInfo.AmsNetID,
					pArrEcConfSlaveInfo := ADR(ConfiguredSlaveInfo),
					cbBufLen			:= SIZEOF(ConfiguredSlaveInfo),
					tTimeout			:= T#1S);

// Init Sequence
CASE InitializeSequence OF
	(* Read Configured Slave Info Data *)
	0:
		GetConfiguredSlaves.bExecute := TRUE;
		IF GetConfiguredSlaves.bBusy THEN
			InitializeSequence := InitializeSequence + 10;
		END_IF

	10:
		IF NOT GetConfiguredSlaves.bBusy AND NOT GetConfiguredSlaves.bError THEN
			CfgSlaveCount := GetConfiguredSlaves.nSlaves;
			IF CfgSlaveCount > Parameter_Diagnostic.ETHERCAT_MASTER_SLAVE_MAX THEN
				Trace('Init Failed - Configured EtherCat Slave amount per master to small! Increase ETHERCAT_MASTER_SLAVE_MAX!');
			ELSE
				InitializeSequence := InitializeSequence + 10;
			END_IF
		END_IF

		IF GetConfiguredSlaves.bError THEN
			_Error := TRUE;
			Trace('Init Failed - Configured EtherCat Slaves could not be read!');
			InitializeSequence := 999;
		END_IF

	20: // Startup time for Ethercat Master	
		StartupTime(IN := TRUE, PT := Parameter_Diagnostic.ETHERCAT_MASTER_START_UP_TIME);
		IF StartupTime.Q THEN
			InitializeSequence := InitializeSequence + 10;
		END_IF

	30:
		Initialize := SUPER^.Initialize();
END_CASE
END_METHOD

METHOD PROTECTED MasterState
VAR_INST
	TypeError			 : BOOL;
	TypeWarning			 : BOOL;
	MasterDevStateString : STRING;
END_VAR
// Read Master state
EcGetMasterDevState(sNetId := _EtherCatMasterInfo.AmsNetID, tTimeout := T#1S, nDevState => MasterDevState);

// Sequence
CASE MasterSeq OF
	(* Wait for start *)
	0:
		EcGetMasterDevState.bExecute := FALSE;

	(* Read Master State*)
	10:
		EcGetMasterDevState.bExecute := TRUE;
		IF EcGetMasterDevState.bBusy THEN
			MasterSeq := MasterSeq + 10;
		END_IF

	20:
		IF NOT EcGetMasterDevState.bBusy AND NOT EcGetMasterDevState.bError THEN
			MasterSeq := MasterSeq + 10;
		END_IF

		IF EcGetMasterDevState.bError THEN
			MasterSeq := 999;
		END_IF

	(* Evaluate Master State *)
	30:
		MasterDevStateString := LookupMasterDevState(State := MasterDevState, TypeError => TypeError, TypeWarning => TypeWarning);
		IF MasterDevState <> 0 THEN
			IF TypeError THEN
				IF NOT MasterAlarms[E_EtherCatMaster.MasterError].bRaised THEN
					SUPER^.RaiseAlarmWithStrings(Alarm := MasterAlarms[E_EtherCatMaster.MasterError], String_1 := MasterDevStateString, String_2 := '');
				END_IF
			END_IF

			IF TypeWarning THEN
				IF NOT MasterAlarms[E_EtherCatMaster.MasterWarning].bRaised THEN
					SUPER^.RaiseEventWithStrings(Alarm := MasterAlarms[E_EtherCatMaster.MasterWarning], String_1 := MasterDevStateString, String_2 := '');
				END_IF
			END_IF

			_ErrorID := MasterDevState;
		END_IF

		MasterSeq := MasterSeq + 10;

	40:
		MasterSeq := 0;

	(* Sequence Error*)
	999:
		Trace('FB_Component_EtherCatMaster - Error get Master State Sequence!');
		MasterSeq := 0;
END_CASE
END_METHOD

METHOD PROTECTED SlaveState
VAR_INST
	BitMaskDiag	 : BYTE := 16#0F;
	ErrorSlave	 : BOOL;
	FaultedSlave : UDINT;
	SyncUnit	 : UDINT;

	// Sync Unit Diagnostic
	SlavesInSyncUnitPartA : STRING;
	SlavesInSyncUnitPartB : STRING;
END_VAR
{analysis -14}
{analysis -07}
{analysis -19}

// Get slave topology info
GetSlaveTopologyInfo(sNetId	  := _EtherCatMasterInfo.AmsNetID,
					 pAddrBuf := ADR(EcSlaveTopologyInfo),
					 cbBufLen := SIZEOF(EcSlaveTopologyInfo),
					 tTimeout := T#5S);

// Get all slave states
EcGetAllSlaveStates(sNetId	  := _EtherCatMasterInfo.AmsNetID,
					pStateBuf := ADR(EcSlavesState),
					cbBufLen  := SIZEOF(EcSlavesState),
					tTimeout  := T#5S);

// Sequence
CASE SlaveSeq OF
	(* Wait for start *)
	0:
		EcGetAllSlaveStates.bExecute  := FALSE;
		GetConfiguredSlaves.bExecute  := FALSE;
		GetSlaveTopologyInfo.bExecute := FALSE;

	(* Update Topology*)
	10:
		GetSlaveTopologyInfo.bExecute := TRUE;
		IF GetSlaveTopologyInfo.bBusy THEN
			SlaveSeq := SlaveSeq + 10;
		END_IF

	20:
		IF NOT GetSlaveTopologyInfo.bBusy AND NOT GetSlaveTopologyInfo.bError THEN
			SlaveSeq := SlaveSeq + 10;
		END_IF

		IF GetSlaveTopologyInfo.bError THEN
			SlaveSeq := 999;
		END_IF

	(* Update Sync Units*)
	30:
		ipEtherCatSyncUnits.Update();
		IF ipEtherCatSyncUnits.Busy THEN
			SlaveSeq := SlaveSeq + 10;
		END_IF

	40:
		IF NOT ipEtherCatSyncUnits.Busy AND NOT ipEtherCatSyncUnits.Error THEN
			// Get EtherCat Sync Units
			SyncUnits REF= ipEtherCatSyncUnits.SyncUnits;
			SlaveSeq  := SlaveSeq + 10;
		END_IF

		IF ipEtherCatSyncUnits.Error THEN
			SlaveSeq := 999;
		END_IF

	(* Read Slave States *)
	50:
		EcGetAllSlaveStates.bExecute := TRUE;
		IF EcGetAllSlaveStates.bBusy THEN
			SlaveSeq := SlaveSeq + 10;
		END_IF

	60:
		IF NOT EcGetAllSlaveStates.bBusy AND NOT EcGetAllSlaveStates.bError THEN
			SlaveCount := EcGetAllSlaveStates.nSlaves;
			SlaveSeq   := SlaveSeq + 10;
		END_IF

		IF EcGetAllSlaveStates.bError THEN
			SlaveSeq := 999;
		END_IF

	(* Evaluate Slave Error *)
	70:
		FOR FaultedSlave := 0 TO (CfgSlaveCount - 1) DO
			// Slave State
			IF (EcSlavesState[FaultedSlave].deviceState AND BitMaskDiag) <> EC_DEVICE_STATE_OP AND EcSlaveTopologyInfo[FaultedSlave].nStatusBits.4 = FALSE THEN
				IF EcSlavesState[FaultedSlave].deviceState.7 THEN // Slave is Disabled or hot connect- warning only
					THIS^.RaiseWarningWithStringParameters(Warning	:= SlaveWarnings[FaultedSlave],
														   String_1 := SlaveWarnings[FaultedSlave].ipSourceInfo.sName,
														   String_2 := LookupSlaveDevState(FaultedSlave),
														   String_3 := '');
				ELSE
					THIS^.RaiseAlarmWithStringsAndFlags(Alarm	 := SlaveErrors[FaultedSlave],
														String_1 := SlaveErrors[FaultedSlave].ipSourceInfo.sName,
														String_2 := LookupSlaveDevState(FaultedSlave),
														String_3 := '');

					ErrorSlave := TRUE;
				END_IF
			END_IF

			// Slave Linking Error
			IF (EcSlavesState[FaultedSlave].linkState AND BitMaskDiag) <> EC_LINK_STATE_OK AND EcSlaveTopologyInfo[FaultedSlave].nStatusBits.4 = FALSE THEN
				THIS^.RaiseAlarmWithStringsAndFlags(Alarm	 := SlaveErrors[FaultedSlave],
													String_1 := SlaveErrors[FaultedSlave].ipSourceInfo.sName,
													String_2 := LookupSlaveDevState(FaultedSlave),
													String_3 := '');
			END_IF

			// Raise related Sync Unit Alarm
			FOR SyncUnit := 1 TO Parameter_Diagnostic.ETHERCAT_MASTER_SYNC_UNIT_MAX DO
				IF SyncUnits[SyncUnit].Parent = THIS^.Name THEN
					IF SlaveIsPartOfSyncUnit(SlaveAddr := ConfiguredSlaveInfo[FaultedSlave].nAddr, SyncUnit := SyncUnits[SyncUnit]) AND SlaveErrors[FaultedSlave].bRaised OR SlaveWarnings[FaultedSlave].bRaised THEN
						THIS^.GetSyncUnitSlaveNames(SyncUnit := SyncUnits[SyncUnit], SlavesInSyncUnitPartA => SlavesInSyncUnitPartA, SlavesInSyncUnitPartB => SlavesInSyncUnitPartB);
						THIS^.RaiseWarningWithStringParameters(Warning	:= SyncUnitWarnings[SyncUnit],
															   String_1 := CONCAT(SyncUnits[SyncUnit].Parent, CONCAT(' - ', SyncUnits[SyncUnit].Name)),
															   String_2 := SlavesInSyncUnitPartA,
															   String_3 := SlavesInSyncUnitPartB);

						EXIT;
					END_IF
				END_IF
			END_FOR
		END_FOR

		SlaveSeq := SlaveSeq + 10;

	80:
		SlaveSeq := 0;

	(* Sequence Error*)
	999:
		Trace('FB_Component_EtherCatMaster - Error get Slave States Sequence!');
		SlaveSeq := 0;
END_CASE
END_METHOD

PROPERTY EtherCatMasterInfo : REFERENCE TO ST_DeviceInfo
SET
{analysis -21}
_EtherCatMasterInfo REF= EtherCatMasterInfo;
END_SET
END_PROPERTY

END_FUNCTION_BLOCK

// EtherCat Diagnostic/F_EtherCAT_VendorIDtoString
FUNCTION F_EtherCAT_VendorIDtoString : STRING(255)
VAR_INPUT
	VendorId : UDINT;
END_VAR

CASE VendorID OF
	16#00000001:
		F_EtherCAT_VendorIDtoString := 'EtherCAT Technology Group';

	16#00000002:
		F_EtherCAT_VendorIDtoString := 'Beckhoff Automation GmbH & Co. KG';

	16#00000003:
		F_EtherCAT_VendorIDtoString := 'Scuola Superiore SantAnna, PERCRO';

	16#00000004:
		F_EtherCAT_VendorIDtoString := 'HMS Technology Center Ravensburg GmbH';

	16#00000005:
		F_EtherCAT_VendorIDtoString := 'Vector Informatik GmbH';

	16#00000006:
		F_EtherCAT_VendorIDtoString := 'KNESTEL Technologie & Elektronik GmbH';

	16#00000007:
		F_EtherCAT_VendorIDtoString := 'Janz Tec AG';

	16#00000009:
		F_EtherCAT_VendorIDtoString := 'Shenyang Jinchi Chuangxin Technology Co.,LTD';

	16#0000000A:
		F_EtherCAT_VendorIDtoString := 'CMZ Sistemi Elettronici S.r.l.';

	16#0000000B:
		F_EtherCAT_VendorIDtoString := 'JSL Technology Co.,Ltd';

	16#0000000C:
		F_EtherCAT_VendorIDtoString := 'comemso GmbH';

	16#0000000D:
		F_EtherCAT_VendorIDtoString := 'Softing Industrial Automation GmbH';

	16#0000000E:
		F_EtherCAT_VendorIDtoString := 'MicroControl GmbH & Co. KG';

	16#0000000F:
		F_EtherCAT_VendorIDtoString := 'ESR Pollmeier GmbH';

	16#00000010:
		F_EtherCAT_VendorIDtoString := 'Beihang University, School of Mechanical Engineering & Automation';

	16#00000011:
		F_EtherCAT_VendorIDtoString := 'GKG Precision Machine Co., Ltd.';

	16#00000012:
		F_EtherCAT_VendorIDtoString := 'Inatech Co., Ltd.';

	16#00000013:
		F_EtherCAT_VendorIDtoString := 'Fritz Kubler GmbH';

	16#00000014:
		F_EtherCAT_VendorIDtoString := 'KEB Automation KG';

	16#00000015:
		F_EtherCAT_VendorIDtoString := 'AJINEXTEK Co. Ltd.';

	16#00000016:
		F_EtherCAT_VendorIDtoString := 'KEBA Industrial Automation Germany GmbH';

	16#00000017:
		F_EtherCAT_VendorIDtoString := 'esd electronics gmbh';

	16#00000018:
		F_EtherCAT_VendorIDtoString := 'M2I Corporation';

	16#00000019:
		F_EtherCAT_VendorIDtoString := 'NSD Corporation';

	16#0000001A:
		F_EtherCAT_VendorIDtoString := 'Shanghai ECAT Science and Technology Co.,Ltd';

	16#0000001B:
		F_EtherCAT_VendorIDtoString := 'HMS Industrial Networks AB';

	16#0000001C:
		F_EtherCAT_VendorIDtoString := 'epis Automation GmbH & Co. KG';

	16#0000001D:
		F_EtherCAT_VendorIDtoString := 'Festo SE & Co. KG';

	16#0000001E:
		F_EtherCAT_VendorIDtoString := 'Shanghai MicroPort Medical (Group) Co., Ltd.';

	16#00000020:
		F_EtherCAT_VendorIDtoString := 'DST Robot Co. Ltd.';

	16#00000021:
		F_EtherCAT_VendorIDtoString := 'WAGO GmbH & Co. KG';

	16#00000022:
		F_EtherCAT_VendorIDtoString := 'Wuhan Farley Laserlab Cutting Welding System Engineering Co., Ltd.';

	16#00000023:
		F_EtherCAT_VendorIDtoString := 'ACTi Corporation';

	16#00000024:
		F_EtherCAT_VendorIDtoString := 'Bosch Rexroth AG';

	16#00000025:
		F_EtherCAT_VendorIDtoString := 'Inexbot NanJing Technology Co., Ltd.';

	16#00000026:
		F_EtherCAT_VendorIDtoString := 'Hongke Technology Co., Ltd.';

	16#00000027:
		F_EtherCAT_VendorIDtoString := 'Selcom Group S.p.A.';

	16#00000028:
		F_EtherCAT_VendorIDtoString := 'Moog GmbH';

	16#00000029:
		F_EtherCAT_VendorIDtoString := 'INTEC - Motion Systems GmbH';

	16#0000002A:
		F_EtherCAT_VendorIDtoString := 'HIGHYAG Lasertechnologie GmbH';

	16#0000002B:
		F_EtherCAT_VendorIDtoString := 'Doosan Robotics Inc.';

	16#0000002C:
		F_EtherCAT_VendorIDtoString := 'Probot Automation GmbH';

	16#0000002D:
		F_EtherCAT_VendorIDtoString := 'Beijing NiMotion Control Technology Co., Ltd.';

	16#0000002E:
		F_EtherCAT_VendorIDtoString := 'Dinkle Enterprise Co. Ltd.';

	16#0000002F:
		F_EtherCAT_VendorIDtoString := 'Guangzhou Kossi Intelligent Technology Co., Ltd.';

	16#00000030:
		F_EtherCAT_VendorIDtoString := 'Epec Oy';

	16#00000031:
		F_EtherCAT_VendorIDtoString := 'Chengdu EVControl Technology Co., Ltd.';

	16#00000032:
		F_EtherCAT_VendorIDtoString := 'Robotek Otomasyon Teknolojileri San. Tic. Ltd. Sti.';

	16#00000033:
		F_EtherCAT_VendorIDtoString := 'Shenzhen Liwi Automation Co., Ltd.';

	16#00000034:
		F_EtherCAT_VendorIDtoString := 'port industrial automation GmbH';

	16#00000035:
		F_EtherCAT_VendorIDtoString := 'Weissler Information Technology GmbH';

	16#00000036:
		F_EtherCAT_VendorIDtoString := 'FAS Electronics (Fujian) Co.,LTD.';

	16#00000037:
		F_EtherCAT_VendorIDtoString := 'Guangzhou Honest Automation Co., Ltd.';

	16#00000038:
		F_EtherCAT_VendorIDtoString := 'InCAT';

	16#00000039:
		F_EtherCAT_VendorIDtoString := 'Burkert Werke GmbH & Co. KG';

	16#0000003A:
		F_EtherCAT_VendorIDtoString := 'Adtec Plasma Technology Co. Ltd.';

	16#0000003B:
		F_EtherCAT_VendorIDtoString := 'Lenze SE';

	16#0000003C:
		F_EtherCAT_VendorIDtoString := 'Shanghai 3cRobot Co.,Ltd.';

	16#0000003D:
		F_EtherCAT_VendorIDtoString := 'Tianjin Fuyun Tianyi Technology Co., Ltd.';

	16#0000003E:
		F_EtherCAT_VendorIDtoString := 'MH Robot & Automation Co., Ltd.';

	16#0000003F:
		F_EtherCAT_VendorIDtoString := 'Weihai IDENCODER Electronic Technology Co.,Ltd';

	16#00000040:
		F_EtherCAT_VendorIDtoString := 'Temposonics GmbH & Co. KG';

	16#00000041:
		F_EtherCAT_VendorIDtoString := 'HIOKI E.E. Corporation';

	16#00000042:
		F_EtherCAT_VendorIDtoString := 'TIGRIS Elektronik GmbH';

	16#00000043:
		F_EtherCAT_VendorIDtoString := 'Hangzhou Muxun Technology Co., Ltd.';

	16#00000044:
		F_EtherCAT_VendorIDtoString := 'Hilscher Gesellschaft fur Systemautomation mbH';

	16#00000045:
		F_EtherCAT_VendorIDtoString := 'MINTROBOT Co., Ltd.';

	16#00000046:
		F_EtherCAT_VendorIDtoString := 'Bosch Rexroth (Xi’an) Electric Drives and Controls Co., Ltd.';

	16#00000047:
		F_EtherCAT_VendorIDtoString := 'WIKA Alexander Wiegand SE & Co. KG';

	16#00000048:
		F_EtherCAT_VendorIDtoString := 'Handtmann e-solutions GmbH & Co. KG';

	16#00000049:
		F_EtherCAT_VendorIDtoString := 'Industrial Software Co.';

	16#0000004A:
		F_EtherCAT_VendorIDtoString := 'Henschel-Robotics GmbH';

	16#0000004B:
		F_EtherCAT_VendorIDtoString := 'Ever Elettronica srl';

	16#0000004C:
		F_EtherCAT_VendorIDtoString := 'Smart Motion Control Co., Ltd.';

	16#0000004D:
		F_EtherCAT_VendorIDtoString := 'EZMotion Technologies, Inc';

	16#0000004E:
		F_EtherCAT_VendorIDtoString := 'Xeryon bvba';

	16#0000004F:
		F_EtherCAT_VendorIDtoString := 'Murrelektronik GmbH';

	16#00000050:
		F_EtherCAT_VendorIDtoString := 'Orion Technology Co., Ltd.';

	16#00000051:
		F_EtherCAT_VendorIDtoString := 'e.con power solutions GmbH';

	16#00000052:
		F_EtherCAT_VendorIDtoString := 'Beijing Jingwei New Technology Textile Machinery CO., LTD.';

	16#00000053:
		F_EtherCAT_VendorIDtoString := 'Delta Farm Co., Ltd.';

	16#00000054:
		F_EtherCAT_VendorIDtoString := 'Quick Tech Japan LTD.';

	16#00000055:
		F_EtherCAT_VendorIDtoString := 'BBK Test Systems Co.,Ltd';

	16#00000057:
		F_EtherCAT_VendorIDtoString := 'Komax AG';

	16#00000058:
		F_EtherCAT_VendorIDtoString := 'Shanghai Fangling Software Co., Ltd.';

	16#00000059:
		F_EtherCAT_VendorIDtoString := 'SEW-EURODRIVE GmbH & Co KG';

	16#0000005A:
		F_EtherCAT_VendorIDtoString := 'Shenzhen Yoda Motion Control Technology Co., Ltd.';

	16#0000005C:
		F_EtherCAT_VendorIDtoString := 'Surface Generation Ltd';

	16#0000005D:
		F_EtherCAT_VendorIDtoString := 'Schleicher Electronic Berlin GmbH';

	16#0000005E:
		F_EtherCAT_VendorIDtoString := 'Creator Industry (Suzhou) Co., Ltd.';

	16#0000005F:
		F_EtherCAT_VendorIDtoString := 'Baumer Electric AG';

	16#00000060:
		F_EtherCAT_VendorIDtoString := 'INCAA Computers BV';

	16#00000061:
		F_EtherCAT_VendorIDtoString := 'Guangdong Sygole Intelligent Technology Co., Ltd.';

	16#00000062:
		F_EtherCAT_VendorIDtoString := 'Bachmann electronic GmbH';

	16#00000063:
		F_EtherCAT_VendorIDtoString := 'Changsha BSL Info. Tech. Co., Ltd.';

	16#00000064:
		F_EtherCAT_VendorIDtoString := 'XPrecise (Beijing) Medical Technology Co., Ltd.';

	16#00000065:
		F_EtherCAT_VendorIDtoString := 'Beijing Surgerii Robotics Company Limited';

	16#00000066:
		F_EtherCAT_VendorIDtoString := 'ROFIN-SINAR Laser GmbH';

	16#00000067:
		F_EtherCAT_VendorIDtoString := 'MAC Valves, Inc.';

	16#00000068:
		F_EtherCAT_VendorIDtoString := 'Fagor Automation Sociedad Cooperativa';

	16#0000006A:
		F_EtherCAT_VendorIDtoString := 'KOLLMORGEN Corporation';

	16#0000006B:
		F_EtherCAT_VendorIDtoString := 'Woodward Kempen GmbH';

	16#0000006C:
		F_EtherCAT_VendorIDtoString := 'B&R Industrial Automation GmbH';

	16#0000006D:
		F_EtherCAT_VendorIDtoString := 'Shenzhen Konghui Intellitech Co.,Ltd.';

	16#0000006E:
		F_EtherCAT_VendorIDtoString := 'AutoLink Electronics (ShenZhen) Co., Ltd.';

	16#00000070:
		F_EtherCAT_VendorIDtoString := 'MIRAPRO Co., Ltd.';

	16#00000072:
		F_EtherCAT_VendorIDtoString := 'INAMCT CO.,LTD.';

	16#00000073:
		F_EtherCAT_VendorIDtoString := 'Global Automation AB';

	16#00000075:
		F_EtherCAT_VendorIDtoString := 'WONIK IPS Co., LTD';

	16#00000077:
		F_EtherCAT_VendorIDtoString := 'SLC Sautter Lift Components GmbH & Co. KG';

	16#00000079:
		F_EtherCAT_VendorIDtoString := 'ETLsoft Kft.';

	16#0000007A:
		F_EtherCAT_VendorIDtoString := 'SIBONAC Laser Technologies Co.,Ltd.';

	16#0000007B:
		F_EtherCAT_VendorIDtoString := 'TUV SUD Rail GmbH';

	16#0000007F:
		F_EtherCAT_VendorIDtoString := 'Shanghai Synrize Automatic Co., Ltd.';

	16#00000080:
		F_EtherCAT_VendorIDtoString := 'YDIIT Co., Ltd.';

	16#00000081:
		F_EtherCAT_VendorIDtoString := 'AUBO (BEIJING) ROBOTICS TECHNOLOGY CO., LTD';

	16#00000082:
		F_EtherCAT_VendorIDtoString := 'Infranor SAS';

	16#00000083:
		F_EtherCAT_VendorIDtoString := 'OMRON Corporation';

	16#00000084:
		F_EtherCAT_VendorIDtoString := 'Phoenix Contact GmbH & Co. KG';

	16#00000087:
		F_EtherCAT_VendorIDtoString := 'Boneng Transmission Co. Ltd.';

	16#00000088:
		F_EtherCAT_VendorIDtoString := 'THINKVO Automation Equipment Co.,Ltd.';

	16#00000089:
		F_EtherCAT_VendorIDtoString := 'Shenyang Jinchi Chuangxin Technology Co.,LTD';

	16#0000008A:
		F_EtherCAT_VendorIDtoString := 'System Ceramics S.p.A.';

	16#0000008E:
		F_EtherCAT_VendorIDtoString := 'Lazer Safe Pty Ltd';

	16#00000090:
		F_EtherCAT_VendorIDtoString := 'Vacon Oy';

	16#00000093:
		F_EtherCAT_VendorIDtoString := 'Gefran S.P.A.';

	16#00000094:
		F_EtherCAT_VendorIDtoString := 'RSV Romanski Sensor- und Verstarkertechnik GmbH';

	16#00000097:
		F_EtherCAT_VendorIDtoString := 'Camozzi Automation S.p.A.';

	16#00000099:
		F_EtherCAT_VendorIDtoString := 'COTRUST TECHNOLOGIES CO., LTD.';

	16#0000009A:
		F_EtherCAT_VendorIDtoString := 'Elmo Motion Control Ltd.';

	16#0000009B:
		F_EtherCAT_VendorIDtoString := 'Hope Win Industrial Co.,Ltd.';

	16#0000009C:
		F_EtherCAT_VendorIDtoString := 'Hans Turck GmbH & Co. KG';

	16#0000009F:
		F_EtherCAT_VendorIDtoString := 'Konsept Elektronik Otomasyon ve Yazilim';

	16#000000A0:
		F_EtherCAT_VendorIDtoString := 'Sontheim Industrie Elektronik GmbH';

	16#000000A2:
		F_EtherCAT_VendorIDtoString := 'HORIBA STEC, Co., Ltd.';

	16#000000A3:
		F_EtherCAT_VendorIDtoString := 'HORIBA Instruments Incorporated';

	16#000000A4:
		F_EtherCAT_VendorIDtoString := 'HORIBA Precision Instruments (Beijing) Co,.Ltd.';

	16#000000A5:
		F_EtherCAT_VendorIDtoString := 'Hirschmann Automation and Control GmbH';

	16#000000A6:
		F_EtherCAT_VendorIDtoString := 'Actuated Robots Ltd';

	16#000000A7:
		F_EtherCAT_VendorIDtoString := 'Wieland Electric GmbH';

	16#000000AA:
		F_EtherCAT_VendorIDtoString := 'Beijing A&E Technologies Co., Ltd.';

	16#000000AB:
		F_EtherCAT_VendorIDtoString := 'Copley Controls, a Division of Analogic Corporation';

	16#000000AC:
		F_EtherCAT_VendorIDtoString := 'Atlas Copco IAS GmbH';

	16#000000AD:
		F_EtherCAT_VendorIDtoString := 'Pepperl+Fuchs SE';

	16#000000AF:
		F_EtherCAT_VendorIDtoString := 'Johannes Hubner Fabrik elektrischer Maschinen GmbH';

	16#000000B1:
		F_EtherCAT_VendorIDtoString := 'Bristol Industrial & Research Associates Ltd';

	16#000000B3:
		F_EtherCAT_VendorIDtoString := 'Bucher Automation AG';

	16#000000B4:
		F_EtherCAT_VendorIDtoString := 'Rob Surgical Systems S.L.';

	16#000000B7:
		F_EtherCAT_VendorIDtoString := 'ABB Oy';

	16#000000B9:
		F_EtherCAT_VendorIDtoString := 'STOBER Antriebstechnik GmbH + Co. KG';

	16#000000BB:
		F_EtherCAT_VendorIDtoString := 'Shanghai Baobin Robot Automation Technology CO., LTD.';

	16#000000BC:
		F_EtherCAT_VendorIDtoString := 'AEC S.r.l.';

	16#000000BD:
		F_EtherCAT_VendorIDtoString := 'ADVANCED Motion Controls';

	16#000000BE:
		F_EtherCAT_VendorIDtoString := 'Bloom Energy (India) Private Limited';

	16#000000C0:
		F_EtherCAT_VendorIDtoString := 'Technofusion Co.,Ltd.';

	16#000000C5:
		F_EtherCAT_VendorIDtoString := 'Comdel, Inc.';

	16#000000C6:
		F_EtherCAT_VendorIDtoString := 'Mitrol S.r.l.';

	16#000000CC:
		F_EtherCAT_VendorIDtoString := 'DENSAN CO., LTD.';

	16#000000CD:
		F_EtherCAT_VendorIDtoString := 'Wipotec GmbH';

	16#000000CE:
		F_EtherCAT_VendorIDtoString := 'Mitsubishi Electric India Pvt. Ltd.';

	16#000000D5:
		F_EtherCAT_VendorIDtoString := 'Bonfiglioli Deutschland GmbH';

	16#000000D6:
		F_EtherCAT_VendorIDtoString := 'HENSOLDT Optronics GmbH';

	16#000000D9:
		F_EtherCAT_VendorIDtoString := 'Phase Motion Control S.p.A.';

	16#000000DA:
		F_EtherCAT_VendorIDtoString := 'Diener Automation GmbH & Co. KG';

	16#000000DB:
		F_EtherCAT_VendorIDtoString := 'Dorabot Inc.';

	16#000000DD:
		F_EtherCAT_VendorIDtoString := 'Samsung Electro-Mechanics Co., Ltd.';

	16#000000DE:
		F_EtherCAT_VendorIDtoString := 'Dave Engineering LLC';

	16#000000E2:
		F_EtherCAT_VendorIDtoString := 'plating electronic GmbH';

	16#000000E3:
		F_EtherCAT_VendorIDtoString := 'CHONGQING PULSE ROBOT CONTROL SYSTEM CO., LTD.';

	16#000000E4:
		F_EtherCAT_VendorIDtoString := 'Metronix Megerate und Elektronik GmbH';

	16#000000E6:
		F_EtherCAT_VendorIDtoString := 'InnoStar Semiconductor (Shanghai) Co., Ltd.';

	16#000000E9:
		F_EtherCAT_VendorIDtoString := 'Ascon S.p.A.';

	16#000000EA:
		F_EtherCAT_VendorIDtoString := 'ESAB-ATAS GmbH';

	16#000000EB:
		F_EtherCAT_VendorIDtoString := 'Elektrobit Automotive GmbH';

	16#000000EC:
		F_EtherCAT_VendorIDtoString := 'Baumer Germany GmbH & Co. KG';

	16#000000ED:
		F_EtherCAT_VendorIDtoString := 'E.D. Elettronica Dedicata S.r.l.';

	16#000000EE:
		F_EtherCAT_VendorIDtoString := 'Ingenieurburo Dr. Tammo Winkler';

	16#000000EF:
		F_EtherCAT_VendorIDtoString := 'Elcis Encoder S.r.l.';

	16#000000F0:
		F_EtherCAT_VendorIDtoString := 'University of South Australia, Future Industries Institute';

	16#000000F1:
		F_EtherCAT_VendorIDtoString := 'McLaren Group Limited';

	16#000000F2:
		F_EtherCAT_VendorIDtoString := 'GGuangdong University of Technology, Faculty of Materials and Energy';

	16#000000F4:
		F_EtherCAT_VendorIDtoString := 'Atos SpA';

	16#000000F5:
		F_EtherCAT_VendorIDtoString := 'GMTO Corporation';

	16#000000F8:
		F_EtherCAT_VendorIDtoString := 'Shanghai Micron Automation Co. Ltd.';

	16#000000F9:
		F_EtherCAT_VendorIDtoString := 'Nidec Control Techniques Ltd.';

	16#000000FB:
		F_EtherCAT_VendorIDtoString := 'maxon motor ag';

	16#000000FC:
		F_EtherCAT_VendorIDtoString := 'Yacoub Automation GmbH';

	16#000000FE:
		F_EtherCAT_VendorIDtoString := 'Precitec GmbH & Co. KG';

	16#000000FF:
		F_EtherCAT_VendorIDtoString := 'South China University of Technology';

	16#00000100:
		F_EtherCAT_VendorIDtoString := 'Easydur Italiana di Renato Affri';

	16#00000101:
		F_EtherCAT_VendorIDtoString := 'ISAC Srl.';

	16#00000104:
		F_EtherCAT_VendorIDtoString := 'LMD GmbH';

	16#00000105:
		F_EtherCAT_VendorIDtoString := 'Microcyber Corporation';

	16#00000107:
		F_EtherCAT_VendorIDtoString := 'Nanjing Command Robot Technology Co.,Ltd';

	16#0000010A:
		F_EtherCAT_VendorIDtoString := 'WITTENSTEIN cyber motor GmbH';

	16#0000010B:
		F_EtherCAT_VendorIDtoString := 'WITTENSTEIN motion control GmbH';

	16#0000010D:
		F_EtherCAT_VendorIDtoString := 'TWK-Elektronik GmbH';

	16#0000010F:
		F_EtherCAT_VendorIDtoString := 'PSA Elettronica di F. Grifa';

	16#00000110:
		F_EtherCAT_VendorIDtoString := 'Maxphotonics Co.,Ltd.';

	16#00000111:
		F_EtherCAT_VendorIDtoString := 'HEITEC AG';

	16#00000112:
		F_EtherCAT_VendorIDtoString := 'KALYSTA Actuation SAS';

	16#00000113:
		F_EtherCAT_VendorIDtoString := 'Soft Service Co., Ltd.';

	16#00000114:
		F_EtherCAT_VendorIDtoString := 'SMC Corporation';

	16#00000116:
		F_EtherCAT_VendorIDtoString := 'Eckelmann AG';

	16#00000117:
		F_EtherCAT_VendorIDtoString := 'JVL Industri Elektronik A/S';

	16#00000118:
		F_EtherCAT_VendorIDtoString := 'Hangzhou Liwei Technology Co. LTD.';

	16#0000011C:
		F_EtherCAT_VendorIDtoString := 'ATESTEO GmbH & Co. KG';

	16#0000011D:
		F_EtherCAT_VendorIDtoString := 'Hottinger Bruel & Kjaer GmbH';

	16#00000121:
		F_EtherCAT_VendorIDtoString := 'Leuze electronic GmbH + Co. KG';

	16#00000123:
		F_EtherCAT_VendorIDtoString := 'WEG Drives & Controls - Automacao Ltda';

	16#00000126:
		F_EtherCAT_VendorIDtoString := 'JUMO GmbH & Co. KG';

	16#00000128:
		F_EtherCAT_VendorIDtoString := 'Hans Smart Control Technology Co., Ltd.';

	16#00000129:
		F_EtherCAT_VendorIDtoString := 'HSD S.p.A';

	16#0000012B:
		F_EtherCAT_VendorIDtoString := 'Digital Electronics Corporation';

	16#0000012E:
		F_EtherCAT_VendorIDtoString := 'Lika Electronic Srl';

	16#0000012F:
		F_EtherCAT_VendorIDtoString := 'CSM Computer-Systeme-Messtechnik GmbH';

	16#00000130:
		F_EtherCAT_VendorIDtoString := 'Jihua Laboratory Intelligent Robot Engineering Research Center';

	16#00000135:
		F_EtherCAT_VendorIDtoString := 'DUOmetric AG';

	16#00000137:
		F_EtherCAT_VendorIDtoString := 'Fenwal Controls of Japan,Ltd.';

	16#00000139:
		F_EtherCAT_VendorIDtoString := 'BOSENSE INTELLIGENT CONTROL TECHNOLOGY CO., LTD.';

	16#00000140:
		F_EtherCAT_VendorIDtoString := 'American Rheinmetall Systems, LLC';

	16#00000142:
		F_EtherCAT_VendorIDtoString := 'SCAIME S.A.S.';

	16#00000144:
		F_EtherCAT_VendorIDtoString := 'TECNOLOGIX Srl';

	16#00000146:
		F_EtherCAT_VendorIDtoString := 'LPKF SolarQuipment GmbH';

	16#00000147:
		F_EtherCAT_VendorIDtoString := 'Dr. Fritz Faulhaber GmbH & Co. KG';

	16#00000149:
		F_EtherCAT_VendorIDtoString := 'Fraunhofer-Institut fur Produktionsanlagen und Konstruktionstechnik IPK';

	16#0000014A:
		F_EtherCAT_VendorIDtoString := 'imc Test & Measurement GmbH';

	16#0000014F:
		F_EtherCAT_VendorIDtoString := 'TMG Technologie Management Gruppe Technologie und Engineering GmbH';

	16#00000150:
		F_EtherCAT_VendorIDtoString := 'Shanghai DriveDream Machinery Equipment Co., Ltd.';

	16#00000151:
		F_EtherCAT_VendorIDtoString := 'Zaklad Produkcji Urzadzen Automatyki Sp. z o.o.';

	16#00000152:
		F_EtherCAT_VendorIDtoString := 'Eckelmann FCS GmbH';

	16#00000155:
		F_EtherCAT_VendorIDtoString := 'Bluechips Microhouse Co., Ltd.';

	16#0000015A:
		F_EtherCAT_VendorIDtoString := 'Baumuller Nurnberg GmbH';

	16#0000015B:
		F_EtherCAT_VendorIDtoString := 'ENGEL Elektroantriebe GmbH';

	16#0000015D:
		F_EtherCAT_VendorIDtoString := 'OSRAM GmbH';

	16#0000015E:
		F_EtherCAT_VendorIDtoString := 'Heidrive GmbH';

	16#00000160:
		F_EtherCAT_VendorIDtoString := 'Seltek Ltd.';

	16#00000163:
		F_EtherCAT_VendorIDtoString := 'AeroLas GmbH';

	16#00000165:
		F_EtherCAT_VendorIDtoString := 'Higgs Invention';

	16#00000166:
		F_EtherCAT_VendorIDtoString := 'Valmet Automation Oy';

	16#00000168:
		F_EtherCAT_VendorIDtoString := 'Shanghai AMP&MOONS Automation Co., Ltd.';

	16#00000169:
		F_EtherCAT_VendorIDtoString := 'RINCO ULTRASONICS AG';

	16#0000016A:
		F_EtherCAT_VendorIDtoString := 'Tsubakimoto Chain Co.';

	16#0000016D:
		F_EtherCAT_VendorIDtoString := 'COMSOFT GmbH';

	16#00000170:
		F_EtherCAT_VendorIDtoString := 'Woodward, Inc.';

	16#00000171:
		F_EtherCAT_VendorIDtoString := 'Prima Electro S.p.A.';

	16#00000172:
		F_EtherCAT_VendorIDtoString := 'Fraunhofer-Institut fur Produktionsanlagen und Konstruktionstechnik IPK';

	16#00000173:
		F_EtherCAT_VendorIDtoString := 'Korea Aerospace University';

	16#00000175:
		F_EtherCAT_VendorIDtoString := 'Massachusetts Institute of Technology (MIT)';

	16#00000176:
		F_EtherCAT_VendorIDtoString := 'Pipedream Labs, Inc.';

	16#00000178:
		F_EtherCAT_VendorIDtoString := 'Foshan Korter Automatic Precision Measurement & Control Technology Co., Ltd.';

	16#00000179:
		F_EtherCAT_VendorIDtoString := 'Delltouch Technology Co., LTD.';

	16#0000017A:
		F_EtherCAT_VendorIDtoString := 'Pneumax S.p.A.';

	16#0000017D:
		F_EtherCAT_VendorIDtoString := 'Delta Line SA';

	16#0000017F:
		F_EtherCAT_VendorIDtoString := 'R.T.A. S.r.l.';

	16#00000181:
		F_EtherCAT_VendorIDtoString := 'FEV Software and Testing Solutions GmbH';

	16#00000184:
		F_EtherCAT_VendorIDtoString := 'BEI Sensors SAS';

	16#00000186:
		F_EtherCAT_VendorIDtoString := 'Zhejiang University of Technology, College of Information Engineering';

	16#00000187:
		F_EtherCAT_VendorIDtoString := 'Suzhou HYC Technology Co.,Ltd.';

	16#00000188:
		F_EtherCAT_VendorIDtoString := 'Flexiv Robotics Ltd.';

	16#00000189:
		F_EtherCAT_VendorIDtoString := 'Pilz GmbH & Co. KG';

	16#0000018A:
		F_EtherCAT_VendorIDtoString := 'ASA-RT srl';

	16#0000018C:
		F_EtherCAT_VendorIDtoString := 'University of Patras';

	16#00000190:
		F_EtherCAT_VendorIDtoString := 'Promess Incorporated';

	16#00000191:
		F_EtherCAT_VendorIDtoString := 'PROMESS Gesellschaft fur Montage- und Prufsysteme mbH';

	16#00000192:
		F_EtherCAT_VendorIDtoString := 'Matsusada Precision Inc.';

	16#00000194:
		F_EtherCAT_VendorIDtoString := 'Leine & Linde AB';

	16#00000195:
		F_EtherCAT_VendorIDtoString := 'SIKO GmbH';

	16#00000196:
		F_EtherCAT_VendorIDtoString := 'Ningbo Taicen Electronic-Test Technology Co., Ltd.';

	16#00000198:
		F_EtherCAT_VendorIDtoString := 'Automation Modules, Inc.';

	16#0000019B:
		F_EtherCAT_VendorIDtoString := 'SP.EL. srl';

	16#0000019D:
		F_EtherCAT_VendorIDtoString := 'Deutschmann Automation GmbH & Co. KG';

	16#0000019E:
		F_EtherCAT_VendorIDtoString := 'Golden A/S';

	16#000001A1:
		F_EtherCAT_VendorIDtoString := 'Brunner Elektronik AG';

	16#000001A2:
		F_EtherCAT_VendorIDtoString := 'Heckner Electronics GmbH';

	16#000001A3:
		F_EtherCAT_VendorIDtoString := 'TECHNOSOFT S.A.';

	16#000001A4:
		F_EtherCAT_VendorIDtoString := 'Kongsberg Maritime AS';

	16#000001A6:
		F_EtherCAT_VendorIDtoString := 'REO AG';

	16#000001AC:
		F_EtherCAT_VendorIDtoString := 'Kyushu Institute of Technology, Ochi & Kurosaki Lab, School of Computer Science and Systems Engineering';

	16#000001AF:
		F_EtherCAT_VendorIDtoString := 'Yanfeng Automotive Interior Systems Co. Ltd.';

	16#000001B0:
		F_EtherCAT_VendorIDtoString := 'ABB AB, Jokab Safety';

	16#000001B2:
		F_EtherCAT_VendorIDtoString := 'AVENTICS GmbH';

	16#000001B3:
		F_EtherCAT_VendorIDtoString := 'ASCO Numatics GmbH';

	16#000001B4:
		F_EtherCAT_VendorIDtoString := 'Peyer Engineering';

	16#000001B5:
		F_EtherCAT_VendorIDtoString := 'Robox S.P.A.';

	16#000001B8:
		F_EtherCAT_VendorIDtoString := 'PMB Elektronik GmbH';

	16#000001B9:
		F_EtherCAT_VendorIDtoString := 'Sanyo Denki Co., Ltd.';

	16#000001BA:
		F_EtherCAT_VendorIDtoString := 'ZHONGSHAN MLTOR CNC TECHNOLOGY CO., LTD.';

	16#000001BB:
		F_EtherCAT_VendorIDtoString := 'Sciemetric Instruments ULC';

	16#000001BC:
		F_EtherCAT_VendorIDtoString := 'Eurotherm Limited';

	16#000001BD:
		F_EtherCAT_VendorIDtoString := 'Eurotherm Automation SAS';

	16#000001BE:
		F_EtherCAT_VendorIDtoString := 'PRIMES GmbH';

	16#000001C0:
		F_EtherCAT_VendorIDtoString := 'Kobe Steel, Ltd.';

	16#000001C4:
		F_EtherCAT_VendorIDtoString := 'Regatron AG';

	16#000001C7:
		F_EtherCAT_VendorIDtoString := 'Eaton Industries GmbH';

	16#000001D5:
		F_EtherCAT_VendorIDtoString := 'ERGSON GmbH';

	16#000001D8:
		F_EtherCAT_VendorIDtoString := 'Changsha Dynamic Technology Co., Ltd.';

	16#000001DD:
		F_EtherCAT_VendorIDtoString := 'Delta Electronics, Inc.';

	16#000001DF:
		F_EtherCAT_VendorIDtoString := 'Xeikon N.V. - Xeikon Manufacturing and R&D Center';

	16#000001E1:
		F_EtherCAT_VendorIDtoString := 'ASCO L.P.';

	16#000001EB:
		F_EtherCAT_VendorIDtoString := 'AMKmotion GmbH + Co KG';

	16#000001EC:
		F_EtherCAT_VendorIDtoString := 'Plus Electric Co.,Ltd.';

	16#000001EE:
		F_EtherCAT_VendorIDtoString := 'ADTECH (SHENZHEN) CNC TECHNOLOGY CO., LTD.';

	16#000001F4:
		F_EtherCAT_VendorIDtoString := 'Robatech AG';

	16#000001F7:
		F_EtherCAT_VendorIDtoString := 'Industrial Technology Research Institute (ITRI)';

	16#000001F8:
		F_EtherCAT_VendorIDtoString := 'Hunan Lianghu Electromechanical Technology Co., Ltd.';

	16#000001F9:
		F_EtherCAT_VendorIDtoString := 'National Instruments Corporation';

	16#000001FA:
		F_EtherCAT_VendorIDtoString := 'Cavotec Micro-Control AS';

	16#000001FB:
		F_EtherCAT_VendorIDtoString := 'Lafert S.p.A.';

	16#000001FC:
		F_EtherCAT_VendorIDtoString := 'Fernsteuergerate Kurt Oelsch GmbH';

	16#000001FD:
		F_EtherCAT_VendorIDtoString := 'INA - Drives & Mechatronics GmbH & Co. KG';

	16#000001FE:
		F_EtherCAT_VendorIDtoString := 'PRUFTECHNIK NDT GmbH';

	16#000001FF:
		F_EtherCAT_VendorIDtoString := 'Zhejiang Qixing Electron Co., Ltd.';

	16#00000205:
		F_EtherCAT_VendorIDtoString := 'BDF DIGITAL S.p.A.';

	16#00000207:
		F_EtherCAT_VendorIDtoString := 'esitron-electronic GmbH';

	16#00000208:
		F_EtherCAT_VendorIDtoString := 'Weihai New Beiyang Zhengqi Robot Co., Ltd.';

	16#0000020C:
		F_EtherCAT_VendorIDtoString := 'ITOH DENKI CO.,LTD.';

	16#00000210:
		F_EtherCAT_VendorIDtoString := 'iASYS Technology Solution Pvt Ltd.';

	16#00000214:
		F_EtherCAT_VendorIDtoString := 'Kniel System-Electronic GmbH';

	16#00000218:
		F_EtherCAT_VendorIDtoString := 'GERMAN POWER GmbH';

	16#00000219:
		F_EtherCAT_VendorIDtoString := 'Real Time Automation, Inc.';

	16#0000021B:
		F_EtherCAT_VendorIDtoString := 'Swift Engineering, Inc.';

	16#0000021F:
		F_EtherCAT_VendorIDtoString := 'Wachendorff Automation GmbH & Co. KG';

	16#00000222:
		F_EtherCAT_VendorIDtoString := 'IBH-Tec GmbH';

	16#00000223:
		F_EtherCAT_VendorIDtoString := 'Helmholz GmbH & Co. KG';

	16#00000225:
		F_EtherCAT_VendorIDtoString := 'Pantec Engineering AG';

	16#0000022B:
		F_EtherCAT_VendorIDtoString := 'YASKAWA Europe GmbH';

	16#0000022F:
		F_EtherCAT_VendorIDtoString := 'TOKYO KEIKI INC.';

	16#00000230:
		F_EtherCAT_VendorIDtoString := 'Weidmuller Interface GmbH & Co. KG';

	16#00000232:
		F_EtherCAT_VendorIDtoString := 'Kornit Digital Ltd.';

	16#00000233:
		F_EtherCAT_VendorIDtoString := 'Guangdong Xian Jiaotong University Academy';

	16#00000234:
		F_EtherCAT_VendorIDtoString := 'AStepTech (Shenzhen) CNC Co., Ltd.';

	16#0000023A:
		F_EtherCAT_VendorIDtoString := 'ABB AG';

	16#0000023B:
		F_EtherCAT_VendorIDtoString := 'Berghof Automation GmbH';

	16#0000023C:
		F_EtherCAT_VendorIDtoString := 'NS System Co., Ltd.';

	16#0000023D:
		F_EtherCAT_VendorIDtoString := 'Sensor-Technik Wiedemann GmbH';

	16#00000240:
		F_EtherCAT_VendorIDtoString := 'Spezialantriebstechnik GmbH';

	16#00000242:
		F_EtherCAT_VendorIDtoString := 'Agile Robots SE';

	16#00000246:
		F_EtherCAT_VendorIDtoString := 'MKP Co., Ltd.';

	16#00000247:
		F_EtherCAT_VendorIDtoString := 'Harmonic Drive LLC';

	16#0000024B:
		F_EtherCAT_VendorIDtoString := 'Dongguan Kaifull Electronics Technology Co., Ltd.';

	16#0000024E:
		F_EtherCAT_VendorIDtoString := 'Eltex-Elektrostatik-GmbH';

	16#0000024F:
		F_EtherCAT_VendorIDtoString := 'Stotz Feinmesstechnik GmbH';

	16#00000250:
		F_EtherCAT_VendorIDtoString := 'Litens Automotive Partnership';

	16#00000252:
		F_EtherCAT_VendorIDtoString := 'Hilscher North America, Inc.';

	16#00000255:
		F_EtherCAT_VendorIDtoString := 'The Chinese University of Hong Kong, T Stone Robotics Institute';

	16#00000256:
		F_EtherCAT_VendorIDtoString := 'Chengdu CRP Automation Control Technology Co., Ltd.';

	16#00000257:
		F_EtherCAT_VendorIDtoString := 'Dunkermotoren GmbH';

	16#0000025E:
		F_EtherCAT_VendorIDtoString := 'Fuji Electric Co., Ltd.';

	16#0000025F:
		F_EtherCAT_VendorIDtoString := 'Fuji Electric India Private Limited';

	16#00000260:
		F_EtherCAT_VendorIDtoString := 'TRUMPF Huttinger GmbH + Co. KG';

	16#00000265:
		F_EtherCAT_VendorIDtoString := 'Aros Electronics AB';

	16#00000268:
		F_EtherCAT_VendorIDtoString := 'Ho Chi Minh University of Technology, Faculty of Mechanical Engineering';

	16#0000026C:
		F_EtherCAT_VendorIDtoString := 'Nanotec Electronic GmbH & Co. KG';

	16#00000270:
		F_EtherCAT_VendorIDtoString := 'ME-Mesysteme GmbH';

	16#00000275:
		F_EtherCAT_VendorIDtoString := 'Interroll Software & Electronics GmbH';

	16#00000276:
		F_EtherCAT_VendorIDtoString := 'Interroll Innovation GmbH';

	16#00000279:
		F_EtherCAT_VendorIDtoString := 'ISH Ingenieursozietat GmbH';

	16#0000027A:
		F_EtherCAT_VendorIDtoString := 'Moog Unna GmbH';

	16#0000027D:
		F_EtherCAT_VendorIDtoString := 'ebm-papst St. Georgen GmbH & Co. KG';

	16#00000280:
		F_EtherCAT_VendorIDtoString := 'MK Precision Co., Ltd.';

	16#00000283:
		F_EtherCAT_VendorIDtoString := 'Roche Diagnostics AG';

	16#00000284:
		F_EtherCAT_VendorIDtoString := 'Toshiba Schneider Inverter Corporation';

	16#00000285:
		F_EtherCAT_VendorIDtoString := 'Bihl+Wiedemann GmbH';

	16#00000286:
		F_EtherCAT_VendorIDtoString := 'TRINAMIC Motion Control GmbH & Co. KG';

	16#00000288:
		F_EtherCAT_VendorIDtoString := 'Xiangshui Jiayi Electronic Technology Co., Ltd';

	16#00000289:
		F_EtherCAT_VendorIDtoString := 'HDT Srl';

	16#00000291:
		F_EtherCAT_VendorIDtoString := 'Terzo Power Systems, LLC';

	16#00000292:
		F_EtherCAT_VendorIDtoString := 'Horner APG LLC';

	16#00000296:
		F_EtherCAT_VendorIDtoString := 'Performance Motion Devices, Inc.';

	16#00000297:
		F_EtherCAT_VendorIDtoString := 'UNIVER S.p.A.';

	16#0000029A:
		F_EtherCAT_VendorIDtoString := 'C.L.GERHARTL Smart Systems GmbH';

	16#0000029C:
		F_EtherCAT_VendorIDtoString := 'Novanta Technologies Spain S.L.';

	16#0000029D:
		F_EtherCAT_VendorIDtoString := 'CREVIS Co., Ltd.';

	16#000002AA:
		F_EtherCAT_VendorIDtoString := 'WalthMac Measurement & Control Technology Co., Ltd.';

	16#000002AB:
		F_EtherCAT_VendorIDtoString := 'U.I. Lapp GmbH';

	16#000002AD:
		F_EtherCAT_VendorIDtoString := 'NIMAK GmbH';

	16#000002B4:
		F_EtherCAT_VendorIDtoString := 'ELAP S.R.L.';

	16#000002B8:
		F_EtherCAT_VendorIDtoString := 'Gripping Power, Inc.';

	16#000002B9:
		F_EtherCAT_VendorIDtoString := 'Advanced Energy Industries, Inc.';

	16#000002BA:
		F_EtherCAT_VendorIDtoString := 'PBA Systems Pte Ltd';

	16#000002BE:
		F_EtherCAT_VendorIDtoString := 'ORIENTAL MOTOR CO., LTD.';

	16#000002C0:
		F_EtherCAT_VendorIDtoString := 'Glentek, Inc.';

	16#000002C1:
		F_EtherCAT_VendorIDtoString := 'Fronius International GmbH';

	16#000002CE:
		F_EtherCAT_VendorIDtoString := 'SHANGHAI GEMPLE M&E CO.,LTD';

	16#000002D0:
		F_EtherCAT_VendorIDtoString := 'THK Co., Ltd.';

	16#000002D1:
		F_EtherCAT_VendorIDtoString := 'SAMICK THK CO.,LTD.';

	16#000002D3:
		F_EtherCAT_VendorIDtoString := 'Joint Peer Systec Corp.';

	16#000002D8:
		F_EtherCAT_VendorIDtoString := 'halstrup-walcher GmbH';

	16#000002DE:
		F_EtherCAT_VendorIDtoString := 'Trio Motion Technology Ltd.';

	16#000002E1:
		F_EtherCAT_VendorIDtoString := 'Servotronix Motion Control Ltd.';

	16#000002E8:
		F_EtherCAT_VendorIDtoString := 'Suzhou Hualu Industrial Control Technology Co., Ltd.';

	16#000002EA:
		F_EtherCAT_VendorIDtoString := 'Suzhou NODKA Automation Technology Co., Ltd.';

	16#000002EB:
		F_EtherCAT_VendorIDtoString := 'Analytica GmbH';

	16#000002EE:
		F_EtherCAT_VendorIDtoString := 'Metal Work S.p.A';

	16#000002FE:
		F_EtherCAT_VendorIDtoString := 'Shanghai Chaifu Robot Co., Ltd.';

	16#00000300:
		F_EtherCAT_VendorIDtoString := 'Korea Textile Machinery Research Institute (KOTMI)';

	16#00000302:
		F_EtherCAT_VendorIDtoString := 'Digitronic Automationsanlagen GmbH';

	16#00000303:
		F_EtherCAT_VendorIDtoString := 'Dental Manufacturing Unit GmbH';

	16#00000309:
		F_EtherCAT_VendorIDtoString := 'Seowoo Electron CO., LTD.';

	16#0000030C:
		F_EtherCAT_VendorIDtoString := 'LAM Technologies S.a.S.';

	16#0000030E:
		F_EtherCAT_VendorIDtoString := 'IEP Ingenieurburo fur Echtzeitprogrammierung GmbH';

	16#00000311:
		F_EtherCAT_VendorIDtoString := 'Kontron Electronics AG';

	16#00000312:
		F_EtherCAT_VendorIDtoString := 'A-KYUNG Motion Inc.';

	16#00000314:
		F_EtherCAT_VendorIDtoString := 'PI Electronics (H.K.) Ltd.';

	16#00000317:
		F_EtherCAT_VendorIDtoString := 'TOFLO CORPORATION';

	16#00000318:
		F_EtherCAT_VendorIDtoString := 'AXIS CORPORATION';

	16#00000319:
		F_EtherCAT_VendorIDtoString := 'emotas embedded communication GmbH';

	16#0000031D:
		F_EtherCAT_VendorIDtoString := 'Cognex Corporation';

	16#00000320:
		F_EtherCAT_VendorIDtoString := 'Airbus Operations SAS';

	16#00000321:
		F_EtherCAT_VendorIDtoString := 'CODESYS GmbH';

	16#00000325:
		F_EtherCAT_VendorIDtoString := 'SiboTech Automation Co., Ltd.';

	16#00000326:
		F_EtherCAT_VendorIDtoString := 'Intelligent Platforms LLC';

	16#00000327:
		F_EtherCAT_VendorIDtoString := 'ECSPRIME Co., Ltd.';

	16#0000032C:
		F_EtherCAT_VendorIDtoString := 'Guangdong Zhuoli Intelligent Technology Co., LTD';

	16#00000330:
		F_EtherCAT_VendorIDtoString := 'ADVANCE ELECTRIC CO., INC.';

	16#00000331:
		F_EtherCAT_VendorIDtoString := 'SHANGHAI SANY SCIENCE & TECHNOLOGY CO., LTD';

	16#00000333:
		F_EtherCAT_VendorIDtoString := 'HIKARI Co.,Ltd.';

	16#00000334:
		F_EtherCAT_VendorIDtoString := 'CYBELEC S.A.';

	16#00000337:
		F_EtherCAT_VendorIDtoString := 'KOSTAL Industrie Elektrik GmbH';

	16#0000033D:
		F_EtherCAT_VendorIDtoString := 'RS Automation Co., Ltd.';

	16#00000340:
		F_EtherCAT_VendorIDtoString := 'Satelcom Telekomunikasyon, Bilgi ve Iletisim Teknolojileri Ithalat ve Ihracat Sanayi A.S.';

	16#00000343:
		F_EtherCAT_VendorIDtoString := 'K.C.Tech CO.,LTD.';

	16#00000344:
		F_EtherCAT_VendorIDtoString := 'Exlar Corporation';

	16#0000034A:
		F_EtherCAT_VendorIDtoString := 'Dragerwerk AG & Co. KGaA';

	16#0000034C:
		F_EtherCAT_VendorIDtoString := 'Okosis Otomasyon ve Kontrol Sistemleri San. ve Tic. Ltd. Sti.';

	16#0000034D:
		F_EtherCAT_VendorIDtoString := 'Schafer Elektronik GmbH';

	16#0000034E:
		F_EtherCAT_VendorIDtoString := 'Infineon Technologies AG';

	16#00000355:
		F_EtherCAT_VendorIDtoString := 'AIDIN ROBOTICS, INC';

	16#00000358:
		F_EtherCAT_VendorIDtoString := 'Shenzhen Rmotion Technology Co,Ltd.';

	16#00000363:
		F_EtherCAT_VendorIDtoString := 'Analogic Corporation';

	16#00000367:
		F_EtherCAT_VendorIDtoString := 'Novatech-Group Ltd.';

	16#00000368:
		F_EtherCAT_VendorIDtoString := 'Tianjin Geneuo Technology Co.,Ltd.';

	16#00000369:
		F_EtherCAT_VendorIDtoString := 'Kinestas d.o.o.';

	16#0000036D:
		F_EtherCAT_VendorIDtoString := 'HATOX GmbH';

	16#00000373:
		F_EtherCAT_VendorIDtoString := 'TAIAN TECHNOLOGY(WUXI)CO.,LTD.';

	16#0000037F:
		F_EtherCAT_VendorIDtoString := 'XMOS Semiconductor';

	16#00000384:
		F_EtherCAT_VendorIDtoString := 'MKS Denmark ApS';

	16#0000038B:
		F_EtherCAT_VendorIDtoString := 'PLASUS GmbH';

	16#0000038C:
		F_EtherCAT_VendorIDtoString := 'Promicon Elektronik GmbH + Co. KG';

	16#00000397:
		F_EtherCAT_VendorIDtoString := 'Hein Lanz GmbH';

	16#0000039D:
		F_EtherCAT_VendorIDtoString := 'dieEntwickler Elektronik GmbH';

	16#000003AA:
		F_EtherCAT_VendorIDtoString := 'LARsys-Automation GmbH';

	16#000003AB:
		F_EtherCAT_VendorIDtoString := 'Eltronic AG';

	16#000003AD:
		F_EtherCAT_VendorIDtoString := 'Procon Electronics Pty Ltd';

	16#000003AE:
		F_EtherCAT_VendorIDtoString := 'HanYang System';

	16#000003B0:
		F_EtherCAT_VendorIDtoString := 'J. Schneider Elektrotechnik GmbH';

	16#000003B8:
		F_EtherCAT_VendorIDtoString := 'Unitronics LTD';

	16#000003CC:
		F_EtherCAT_VendorIDtoString := 'Motovario S.p.A.';

	16#000003D0:
		F_EtherCAT_VendorIDtoString := 'Wuxi Pneumatic Technical Research Institute Co., Ltd.';

	16#000003D1:
		F_EtherCAT_VendorIDtoString := 'Dongguan Feihu Automation Co., Ltd.';

	16#000003DB:
		F_EtherCAT_VendorIDtoString := 'ABB Motion Ltd.';

	16#000003DC:
		F_EtherCAT_VendorIDtoString := 'Wuxi Lingke Automation Technology Co., Ltd.';

	16#000003E1:
		F_EtherCAT_VendorIDtoString := 'Lite-On Technology Corporation';

	16#000003E3:
		F_EtherCAT_VendorIDtoString := 'Bannari Amman Institute of Technology, Department of Electrical and Electronics Engineering';

	16#000003E7:
		F_EtherCAT_VendorIDtoString := 'AIMOSYSS (Dongguan) Control Technology Co., Ltd.';

	16#000003E9:
		F_EtherCAT_VendorIDtoString := 'Teletec Gesellschaft fur elektronische Systeme mbH';

	16#000003EB:
		F_EtherCAT_VendorIDtoString := 'Stahl GmbH';

	16#000003F3:
		F_EtherCAT_VendorIDtoString := 'CoreTigo Ltd.';

	16#000003F5:
		F_EtherCAT_VendorIDtoString := 'Chieftek Precision Co., Ltd.';

	16#000003FF:
		F_EtherCAT_VendorIDtoString := 'MEXICAN REPS OPERATION S DE RL DE CV (MXRO)';

	16#00000400:
		F_EtherCAT_VendorIDtoString := 'Fenac Teknoloji San. ve Tic. Ltd. Şti.';

	16#00000404:
		F_EtherCAT_VendorIDtoString := 'Applied Motion Products, Inc.';

	16#0000040C:
		F_EtherCAT_VendorIDtoString := 'WITZ Corporation';

	16#00000413:
		F_EtherCAT_VendorIDtoString := 'Shenzhen X-TEC Technology Co., Ltd.';

	16#00000418:
		F_EtherCAT_VendorIDtoString := 'Zume, Inc.';

	16#0000041B:
		F_EtherCAT_VendorIDtoString := 'Shenzhen Zmotion Technology Co., Ltd.';

	16#00000420:
		F_EtherCAT_VendorIDtoString := 'Suzhou Rongsu Technology Co.,Ltd.';

	16#00000428:
		F_EtherCAT_VendorIDtoString := 'TOKKYOKIKI CORPORATION';

	16#0000042B:
		F_EtherCAT_VendorIDtoString := 'TeMec Drive Srl';

	16#00000432:
		F_EtherCAT_VendorIDtoString := 'Peter Huber Kaltemaschinenbau AG';

	16#00000434:
		F_EtherCAT_VendorIDtoString := 'Peter Mess- und Automatisierungstechnik';

	16#0000043C:
		F_EtherCAT_VendorIDtoString := 'Hefei Onsoon Intelligent Electronics Co.,Ltd';

	16#00000441:
		F_EtherCAT_VendorIDtoString := 'Langer & Laumann Ing.-Buro GmbH';

	16#00000442:
		F_EtherCAT_VendorIDtoString := 'EDGESYSTEMS d.o.o.';

	16#00000444:
		F_EtherCAT_VendorIDtoString := 'İlkotek Makine Ve Otomasyon San.Tic.Ltd.Şti';

	16#00000456:
		F_EtherCAT_VendorIDtoString := 'Philips Medical Systems Technologies Ltd.';

	16#00000471:
		F_EtherCAT_VendorIDtoString := 'FURONTEER, INC.';

	16#00000482:
		F_EtherCAT_VendorIDtoString := 'KYOCERA Corporation';

	16#00000483:
		F_EtherCAT_VendorIDtoString := 'EHWA TECHNOLOGIES INFORMATION CO., LTD.';

	16#00000489:
		F_EtherCAT_VendorIDtoString := 'Infinity Sales, Inc.';

	16#0000048A:
		F_EtherCAT_VendorIDtoString := 'OPTON Co.,Ltd.';

	16#000004A2:
		F_EtherCAT_VendorIDtoString := 'UniSwarm SASU';

	16#000004B3:
		F_EtherCAT_VendorIDtoString := 'Pivotal Systems Corporation';

	16#000004B5:
		F_EtherCAT_VendorIDtoString := 'Randy Nurnberger Software und Mikroelektronik';

	16#000004BD:
		F_EtherCAT_VendorIDtoString := 'AMETEK Inc. Haydon Kerk Pittman Division';

	16#000004C1:
		F_EtherCAT_VendorIDtoString := 'IVEK Corporation';

	16#000004C6:
		F_EtherCAT_VendorIDtoString := 'MIDDEX-ELECTRONIC GMBH';

	16#000004CD:
		F_EtherCAT_VendorIDtoString := 'WEETECH GmbH';

	16#000004CE:
		F_EtherCAT_VendorIDtoString := 'Soul&Innovation Ltd.';

	16#000004D2:
		F_EtherCAT_VendorIDtoString := 'Noda Radio Frequency Technologies Co., Ltd.';

	16#000004D5:
		F_EtherCAT_VendorIDtoString := 'Hitachi Information & Telecommunication Engineering, Ltd.';

	16#000004D8:
		F_EtherCAT_VendorIDtoString := 'Microchip Technology Inc.';

	16#000004E2:
		F_EtherCAT_VendorIDtoString := 'M2M craft Co.,Ltd.';

	16#000004F8:
		F_EtherCAT_VendorIDtoString := 'Duplomatic MS S.p.A';

	16#000004F9:
		F_EtherCAT_VendorIDtoString := 'PHYTEC America, LLC';

	16#000004FE:
		F_EtherCAT_VendorIDtoString := 'Shanghai AYAN Industry System Co., Ltd.';

	16#00000500:
		F_EtherCAT_VendorIDtoString := 'Speciaal Machinefabriek Ketels v.o.f.';

	16#00000501:
		F_EtherCAT_VendorIDtoString := 'Beck IPC GmbH';

	16#00000502:
		F_EtherCAT_VendorIDtoString := 'ETAS GmbH';

	16#00000504:
		F_EtherCAT_VendorIDtoString := 'PHYTEC Messtechnik GmbH';

	16#00000505:
		F_EtherCAT_VendorIDtoString := 'ANCA Motion Pty. Ltd';

	16#00000506:
		F_EtherCAT_VendorIDtoString := 'Fachhochschule Koln';

	16#00000507:
		F_EtherCAT_VendorIDtoString := 'IPG Automotive GmbH';

	16#00000508:
		F_EtherCAT_VendorIDtoString := 'Nuvation Engineering Corporation';

	16#00000509:
		F_EtherCAT_VendorIDtoString := 'TR-Electronic GmbH';

	16#0000050A:
		F_EtherCAT_VendorIDtoString := 'Gantner Instruments GmbH';

	16#0000050B:
		F_EtherCAT_VendorIDtoString := 'MKS Instruments Inc.';

	16#0000050C:
		F_EtherCAT_VendorIDtoString := 'ABB AB';

	16#0000050D:
		F_EtherCAT_VendorIDtoString := 'Unitro-Fleischmann';

	16#0000050E:
		F_EtherCAT_VendorIDtoString := 'zub machine control AG';

	16#0000050F:
		F_EtherCAT_VendorIDtoString := 'dSPACE GmbH';

	16#00000510:
		F_EtherCAT_VendorIDtoString := 'Shenzhen ProU software Ltd.';

	16#00000511:
		F_EtherCAT_VendorIDtoString := 'Samsung Heavy Industries';

	16#00000512:
		F_EtherCAT_VendorIDtoString := 'BCE Elektronik GmbH';

	16#00000513:
		F_EtherCAT_VendorIDtoString := 'Jager Computergesteuerte Messtechnik GmbH';

	16#00000514:
		F_EtherCAT_VendorIDtoString := 'avateramedical Mechatronics GmbH';

	16#00000515:
		F_EtherCAT_VendorIDtoString := 'Justek Inc.';

	16#00000516:
		F_EtherCAT_VendorIDtoString := 'Baumer Germany GmbH & Co. KG';

	16#00000517:
		F_EtherCAT_VendorIDtoString := 'Elin EBG Traction GmbH';

	16#00000518:
		F_EtherCAT_VendorIDtoString := 'Meka Robotics';

	16#00000519:
		F_EtherCAT_VendorIDtoString := 'Altera Japan Ltd.';

	16#0000051A:
		F_EtherCAT_VendorIDtoString := 'EBV Elektronik GmbH & Co KG';

	16#0000051B:
		F_EtherCAT_VendorIDtoString := 'Ingenieurgemeinschaft IgH';

	16#0000051C:
		F_EtherCAT_VendorIDtoString := 'IAV GmbH';

	16#0000051D:
		F_EtherCAT_VendorIDtoString := 'Hitachi Industrial Equipment Systems';

	16#0000051E:
		F_EtherCAT_VendorIDtoString := 'TenAsys Corp.';

	16#0000051F:
		F_EtherCAT_VendorIDtoString := 'PONDis AG';

	16#00000520:
		F_EtherCAT_VendorIDtoString := 'Moog Italiana Srl';

	16#00000521:
		F_EtherCAT_VendorIDtoString := 'Walt Disney Imagineering Research & Development, Inc.';

	16#00000522:
		F_EtherCAT_VendorIDtoString := 'Wallner Automation';

	16#00000523:
		F_EtherCAT_VendorIDtoString := 'AVL List GmbH';

	16#00000524:
		F_EtherCAT_VendorIDtoString := 'RITTER-Elektronik GmbH';

	16#00000527:
		F_EtherCAT_VendorIDtoString := 'ZwickRoell GmbH & Co. KG';

	16#00000528:
		F_EtherCAT_VendorIDtoString := 'dresden elektronik ingenieurtechnik gmbh';

	16#00000529:
		F_EtherCAT_VendorIDtoString := 'Tokyo Keiso Co., Ltd.';

	16#0000052C:
		F_EtherCAT_VendorIDtoString := 'Philips Medical Systems (Cleveland) Inc.';

	16#0000052D:
		F_EtherCAT_VendorIDtoString := 'Chess B.V.';

	16#0000052E:
		F_EtherCAT_VendorIDtoString := 'NCT kft';

	16#0000052F:
		F_EtherCAT_VendorIDtoString := 'Anywire Corporation';

	16#00000530:
		F_EtherCAT_VendorIDtoString := 'Shadow Robot Company Ltd.';

	16#00000531:
		F_EtherCAT_VendorIDtoString := 'FeCon GmbH';

	16#00000532:
		F_EtherCAT_VendorIDtoString := 'Fachhochschule Sudwestfalen, Fachbereich Elektrische Energietechnik-Fachgebiet Energieversorgung';

	16#00000533:
		F_EtherCAT_VendorIDtoString := 'add2 Ltd';

	16#00000534:
		F_EtherCAT_VendorIDtoString := 'ARM Automation, Inc.';

	16#00000537:
		F_EtherCAT_VendorIDtoString := 'KNAPP AG';

	16#00000538:
		F_EtherCAT_VendorIDtoString := 'Getriebebau NORD GmbH & Co. KG';

	16#00000539:
		F_EtherCAT_VendorIDtoString := 'Yaskawa Electric Corporation';

	16#0000053A:
		F_EtherCAT_VendorIDtoString := 'OKI IDS Co., Ltd.';

	16#0000053B:
		F_EtherCAT_VendorIDtoString := 'Takasaki Kyoudou Computing Center Co. Ltd.';

	16#0000053C:
		F_EtherCAT_VendorIDtoString := 'NITTETSU ELEX Co., Ltd.';

	16#0000053D:
		F_EtherCAT_VendorIDtoString := 'WACOH-TECH Inc.';

	16#0000053E:
		F_EtherCAT_VendorIDtoString := 'Unjo AB';

	16#0000053F:
		F_EtherCAT_VendorIDtoString := 'Airbus Defence and Space GmbH';

	16#00000540:
		F_EtherCAT_VendorIDtoString := 'ACS Motion Control Ltd.';

	16#00000541:
		F_EtherCAT_VendorIDtoString := 'KEYENCE Corporation';

	16#00000542:
		F_EtherCAT_VendorIDtoString := 'MEFI s.r.o.';

	16#00000543:
		F_EtherCAT_VendorIDtoString := 'm-u-t AG Messgerate fur Medizin- und Umwelttechnik';

	16#00000544:
		F_EtherCAT_VendorIDtoString := 'Universitat Stuttgart, Fakultat Konstruktions-, Produktions- und Fahrzeugtechnik, Institut fur Steuerungstechnik der Werkzeugmaschinen und Fertigungseinrichtungen';

	16#00000545:
		F_EtherCAT_VendorIDtoString := 'ELSENA, Inc.';

	16#00000546:
		F_EtherCAT_VendorIDtoString := 'BE Semiconductor Industries N.V.';

	16#00000547:
		F_EtherCAT_VendorIDtoString := 'Hauni LNI Electronics S.A.';

	16#00000548:
		F_EtherCAT_VendorIDtoString := 'ETEL S.A.';

	16#00000549:
		F_EtherCAT_VendorIDtoString := 'VAT Vakuumventile AG';

	16#0000054A:
		F_EtherCAT_VendorIDtoString := 'LayTec AG';

	16#0000054B:
		F_EtherCAT_VendorIDtoString := 'NUM AG';

	16#0000054C:
		F_EtherCAT_VendorIDtoString := 'Korber Technologies GmbH';

	16#0000054D:
		F_EtherCAT_VendorIDtoString := 'Exatronic, Engenharia Electronica, Lda';

	16#0000054E:
		F_EtherCAT_VendorIDtoString := 'Chinese Academy of Sciences, Institute of Intelligent Machines (IIM)';

	16#0000054F:
		F_EtherCAT_VendorIDtoString := 'Eindhoven University of Technology';

	16#00000550:
		F_EtherCAT_VendorIDtoString := 'Scansonic MI GmbH';

	16#00000551:
		F_EtherCAT_VendorIDtoString := 'Shanghai Sodick Software Co., Ltd.';

	16#00000552:
		F_EtherCAT_VendorIDtoString := 'CHUO ELECTRONICS CO., LTD';

	16#00000553:
		F_EtherCAT_VendorIDtoString := 'Agie Charmilles SA';

	16#00000554:
		F_EtherCAT_VendorIDtoString := 'miControl GmbH';

	16#00000555:
		F_EtherCAT_VendorIDtoString := 'HEIG-VD - Haute Ecole dIngenierie et de Gestion du Canton de Vaud';

	16#00000556:
		F_EtherCAT_VendorIDtoString := 'Wuxi Xinje Electric Co., Ltd.';

	16#00000557:
		F_EtherCAT_VendorIDtoString := 'Jenny Science AG';

	16#00000558:
		F_EtherCAT_VendorIDtoString := 'Industrial Control Communications, Inc.';

	16#00000559:
		F_EtherCAT_VendorIDtoString := 'DMG MORI Additive GmbH';

	16#0000055A:
		F_EtherCAT_VendorIDtoString := 'CKD ELEKTROTECHNIKA, a.s.';

	16#0000055B:
		F_EtherCAT_VendorIDtoString := 'QEM S.r.l.';

	16#0000055C:
		F_EtherCAT_VendorIDtoString := 'Simatex AG';

	16#0000055D:
		F_EtherCAT_VendorIDtoString := 'Kithara Software GmbH';

	16#0000055E:
		F_EtherCAT_VendorIDtoString := 'GE Energy Power Conversion GmbH';

	16#0000055F:
		F_EtherCAT_VendorIDtoString := 'Apparatenfabriek ARA B.V.';

	16#00000560:
		F_EtherCAT_VendorIDtoString := 'Tata Consultancy Services Ltd.';

	16#00000561:
		F_EtherCAT_VendorIDtoString := 'Harmonic Drive Systems Inc.';

	16#00000562:
		F_EtherCAT_VendorIDtoString := 'Tiab Limited';

	16#00000563:
		F_EtherCAT_VendorIDtoString := 'RKC INSTRUMENT INC.';

	16#00000564:
		F_EtherCAT_VendorIDtoString := 'Switched Reluctance Drives Ltd.';

	16#00000566:
		F_EtherCAT_VendorIDtoString := 'AAvnet Electronics Marketing, Inc.';

	16#00000567:
		F_EtherCAT_VendorIDtoString := 'ABB AB';

	16#00000568:
		F_EtherCAT_VendorIDtoString := 'Yamaha Motor Co., Ltd.';

	16#00000569:
		F_EtherCAT_VendorIDtoString := 'KUNBUS GmbH';

	16#0000056A:
		F_EtherCAT_VendorIDtoString := 'ACD Antriebstechnik GmbH';

	16#0000056B:
		F_EtherCAT_VendorIDtoString := 'Bronkhorst High-Tech B.V.';

	16#0000056C:
		F_EtherCAT_VendorIDtoString := 'K.MECS Co., Ltd.';

	16#0000056D:
		F_EtherCAT_VendorIDtoString := 'Ampegon AG';

	16#0000056E:
		F_EtherCAT_VendorIDtoString := 'UFG Elettronica s.r.l.';

	16#0000056F:
		F_EtherCAT_VendorIDtoString := 'Xilinx Inc.';

	16#00000570:
		F_EtherCAT_VendorIDtoString := 'Hitachi Energy Sweden AB';

	16#00000571:
		F_EtherCAT_VendorIDtoString := 'Servoland Corporation';

	16#00000572:
		F_EtherCAT_VendorIDtoString := 'Hivertec, Inc.';

	16#00000573:
		F_EtherCAT_VendorIDtoString := 'Mesa Electronics';

	16#00000574:
		F_EtherCAT_VendorIDtoString := 'OMICRON electronics GmbH';

	16#00000575:
		F_EtherCAT_VendorIDtoString := 'Fike Europe B.v.b.a.';

	16#00000576:
		F_EtherCAT_VendorIDtoString := 'ROPEX Industrie-Elektronik GmbH';

	16#00000577:
		F_EtherCAT_VendorIDtoString := 'TLU - Thuringer Leistungselektronik Union GmbH';

	16#00000579:
		F_EtherCAT_VendorIDtoString := 'Prodrive Technologies B.V.';

	16#0000057A:
		F_EtherCAT_VendorIDtoString := 'miho Inspektionssysteme GmbH';

	16#0000057B:
		F_EtherCAT_VendorIDtoString := 'Tokyo Electron Device Limited';

	16#0000057C:
		F_EtherCAT_VendorIDtoString := 'LINTEC CO., LTD.';

	16#0000057D:
		F_EtherCAT_VendorIDtoString := 'Emhart Glass Vision GmbH';

	16#0000057E:
		F_EtherCAT_VendorIDtoString := 'Seiko Epson Corporation';

	16#0000057F:
		F_EtherCAT_VendorIDtoString := 'ZINSER GmbH';

	16#00000580:
		F_EtherCAT_VendorIDtoString := 'abk-technology GmbH';

	16#00000581:
		F_EtherCAT_VendorIDtoString := 'SUS Corporation';

	16#00000582:
		F_EtherCAT_VendorIDtoString := 'TRsystems GmbH';

	16#00000583:
		F_EtherCAT_VendorIDtoString := 'Harmonic Drive SE';

	16#00000584:
		F_EtherCAT_VendorIDtoString := 'Staubli Faverges SCA';

	16#00000585:
		F_EtherCAT_VendorIDtoString := 'ScienLab electronic systems GmbH';

	16#00000586:
		F_EtherCAT_VendorIDtoString := 'DETO drive systems GmbH';

	16#00000587:
		F_EtherCAT_VendorIDtoString := 'FUJISOFT Incorporated';

	16#00000588:
		F_EtherCAT_VendorIDtoString := 'IAI Corporation';

	16#00000589:
		F_EtherCAT_VendorIDtoString := 'PromAvtomatika';

	16#0000058A:
		F_EtherCAT_VendorIDtoString := 'Kistler Instrumente AG';

	16#0000058B:
		F_EtherCAT_VendorIDtoString := 'LAUDA DR. R. WOBSER GmbH & Co. KG';

	16#0000058C:
		F_EtherCAT_VendorIDtoString := 'Schweitzer Engineering Laboratories, Inc.';

	16#0000058D:
		F_EtherCAT_VendorIDtoString := 'Vital Systems Inc.';

	16#0000058E:
		F_EtherCAT_VendorIDtoString := 'MuTracx International B.V.';

	16#0000058F:
		F_EtherCAT_VendorIDtoString := 'Algo System Co., Ltd.';

	16#00000590:
		F_EtherCAT_VendorIDtoString := 'MB AUTOMATION GmbH & Co. KG';

	16#00000591:
		F_EtherCAT_VendorIDtoString := 'DETO drive systems GmbH';

	16#00000592:
		F_EtherCAT_VendorIDtoString := 'Sealevel Systems, Inc.';

	16#00000593:
		F_EtherCAT_VendorIDtoString := 'igm Robotersysteme AG';

	16#00000594:
		F_EtherCAT_VendorIDtoString := 'WITTENSTEIN electronics GmbH';

	16#00000595:
		F_EtherCAT_VendorIDtoString := 'ZBE Inc.';

	16#00000596:
		F_EtherCAT_VendorIDtoString := 'Zhuhai Yiyao Technology Co., Ltd';

	16#00000597:
		F_EtherCAT_VendorIDtoString := 'Fraunhofer-Institut fur Optronik, Systemtechnik und Bildauswertung, Kompetenzzentrum Industrial Automation (IOSB-INA)';

	16#00000598:
		F_EtherCAT_VendorIDtoString := 'SKF Canada Limited';

	16#00000599:
		F_EtherCAT_VendorIDtoString := 'Galil Motion Control Inc.';

	16#0000059A:
		F_EtherCAT_VendorIDtoString := 'IHI Corporation';

	16#0000059B:
		F_EtherCAT_VendorIDtoString := 'wenglor sensoric gmbh';

	16#0000059C:
		F_EtherCAT_VendorIDtoString := 'Ingeteam Power Technology S.A.';

	16#0000059D:
		F_EtherCAT_VendorIDtoString := 'Texas Instruments Incorporated';

	16#0000059E:
		F_EtherCAT_VendorIDtoString := 'Micro-Vu Corporation';

	16#0000059F:
		F_EtherCAT_VendorIDtoString := 'oehri electronic ag';

	16#000005A0:
		F_EtherCAT_VendorIDtoString := 'Triphase NV';

	16#000005A1:
		F_EtherCAT_VendorIDtoString := 'Glass Soft - Robotica & Sistemas Lda.';

	16#000005A2:
		F_EtherCAT_VendorIDtoString := 'CMR Surgical Ltd.';

	16#000005A3:
		F_EtherCAT_VendorIDtoString := 'China Machinery International Engineering Design & Research Institute CO.,LTD.';

	16#000005A4:
		F_EtherCAT_VendorIDtoString := 'Kastanienbaum GmbH';

	16#000005A5:
		F_EtherCAT_VendorIDtoString := 'HANYOUNG NUX CO., LTD';

	16#000005A6:
		F_EtherCAT_VendorIDtoString := 'SLE quality engineering GmbH & Co. KG';

	16#000005A7:
		F_EtherCAT_VendorIDtoString := 'Omicron NanoTechnology GmbH';

	16#000005A8:
		F_EtherCAT_VendorIDtoString := 'Micromeritics Instrument Corporation';

	16#000005A9:
		F_EtherCAT_VendorIDtoString := 'TRUMPF Laser- und Systemtechnik SE';

	16#000005AB:
		F_EtherCAT_VendorIDtoString := 'Beratron GmbH';

	16#000005AA:
		F_EtherCAT_VendorIDtoString := 'HORIBA Europe GmbH';

	16#000005AC:
		F_EtherCAT_VendorIDtoString := 'Heinz Siegfried AG';

	16#000005AD:
		F_EtherCAT_VendorIDtoString := 'Cebora S.p.A.';

	16#000005AE:
		F_EtherCAT_VendorIDtoString := 'W.E.ST Elektronik GmbH';

	16#000005AF:
		F_EtherCAT_VendorIDtoString := 'ABB AG';

	16#000005B0:
		F_EtherCAT_VendorIDtoString := 'SIEB & MEYER AG';

	16#000005B1:
		F_EtherCAT_VendorIDtoString := 'Harbin Robotics Technology Co., Ltd.';

	16#000005B2:
		F_EtherCAT_VendorIDtoString := 'Protechna Herbst GmbH & Co. KG';

	16#000005B3:
		F_EtherCAT_VendorIDtoString := 'TAEHA Mechatronics Co., Ltd.';

	16#000005B4:
		F_EtherCAT_VendorIDtoString := 'WITTMANN Technology GmbH';

	16#000005B5:
		F_EtherCAT_VendorIDtoString := 'iotec GmbH';

	16#000005B6:
		F_EtherCAT_VendorIDtoString := 'Prodel Technologies';

	16#000005B7:
		F_EtherCAT_VendorIDtoString := 'The Leland Stanford Junior University, Department of Bioengineering';

